# B&R Automation Studio project BatteryControl
Automation Studio 4.9.3.144 SP; technology packages: mapp 5.12.0, mappView 5.12.1

## Configuration Asfordby

CPU X20CP1381, AutomationRuntime A4.26, Build 4.1.2, Safety 0.0, Vc V4.72.2

### Hardware
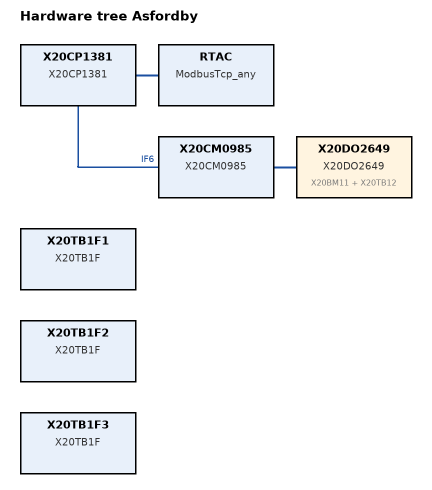
```
RTAC : ModbusTcp_any v1.0.8.0  [ETH1 -> X20CP1381.IF2 (NodeNumber=1) [Cable Type=PowerlinkCable, Length=10, Version=1.0.0.3]]
  IpAddress = 10.71.46.5
  UnitId = 1
  Cb_1
  Cb_1_FunCode = 16
  Cb_1_RefreshTime = 50
  Cb_1_SendMode = 2
  Cb_1_AddrExt = 30
  Cb_1_NumItemsExt = 2
  Cb_1_C_1
  Cb_1_C_1_Name = powerWrite
  Cb_1_C_1_Datatype = 4
  Cb_1_C_1_Dir = 1
  Cb_2
  Cb_2_FunCode = 3
  Cb_2_RefreshTime = 500
  Cb_2_Addr = 10
  Cb_2_C_1
  Cb_2_C_1_Name = operationMode
  Cb_2_C_1_Datatype = 6
  Cb_3
  Cb_3_FunCode = 6
  Cb_3_RefreshTime = 500
  Cb_3_SendMode = 2
  Cb_3_AddrExt = 28
  Cb_3_C_1
  Cb_3_C_1_Name = operationModeWrite
  Cb_3_C_1_Datatype = 6
  Cb_3_C_1_Dir = 1
  Cb_4
  Cb_4_FunCode = 3
  Cb_4_RefreshTime = 500
  Cb_4_Addr = 26
  Cb_4_C_1
  Cb_4_C_1_Name = activePower
  Cb_4_C_1_Datatype = 3
  Cb_5
  Cb_5_FunCode = 3
  Cb_5_RefreshTime = 500
  Cb_5_Addr = 20
  Cb_5_C_1
  Cb_5_C_1_Name = SOC
  Cb_5_C_1_Datatype = 6
X20BM11 : X20BM11 v1.0.0.1 (Disabled=true)  [X2X1 -> X20CM0985.X2X2]
X20CM0985 : X20CM0985 v1.0.6.1  [X2X1 -> X20CP1381.IF6]
  GenRange = 100V
  BusRange = 100V
  Sync1Range = 100V
  Sync2Range = 100V
  CurrentRange = 1A
  UnennSyn = 11000
  UnennGen = 11000
  UnennSamm = 11000
  Inenn = 1250
  Msammel = 10000
  MGen = 10000
  MSyn1 = 10000
  MSyn2 = 10000
  Mstrom = 1250
  TiefpassF = 20
  Ofrequency = 2000
  Ufrequency = 0
  Rfmin = 100
X20CP1381 : X20CP1381 v1.11.0.0  [X1 -> X1.SL; X2 -> X2.SL; X3 -> X3.SL]
  Module X1 (Type=X1, Virtual=true, Version=1.11.0.0)
    Connection (Connector=SS1, TargetModule=X20TB1F1, TargetConnector=SS)
    Connection (Connector=SL, TargetModule=X20CP1381, TargetConnector=X1)
  Module X2 (Type=X2, Virtual=true, Version=1.11.0.0)
    Connection (Connector=SS1, TargetModule=X20TB1F2, TargetConnector=SS)
    Connection (Connector=SL, TargetModule=X20CP1381, TargetConnector=X2)
  Module X3 (Type=X3, Virtual=true, Version=1.11.0.0)
    Connection (Connector=SS1, TargetModule=X20TB1F3, TargetConnector=SS)
    Connection (Connector=SL, TargetModule=X20CP1381, TargetConnector=X3)
  Connector IF2:
    ActivateDevice = 1
    Vnc1
    VncVcObjectName1 = Visu
    VncKeyMappingFile1 = VC\PS2-Keyboard.dis
    VncRefreshRate1 = 500
    VncTitle1 = Debug
    ActivateModbus = 1
    NumSlaves = -1
    NumAllBlocks = -1
    MemSizeIn = -1
    MemSizeOut = -1
  Connector IF3:
    DNAConfiguration = manual
  ConfigurationID = Static_Config1
  TimerDeviceType = SWIOTIMER
  SystemTick = 5000
  IdleTaskClass = 4
  Cyclic1Duration = 5000
  Cyclic1Tolerance = 5000
  Cyclic2Duration = 10000
  Cyclic2Tolerance = 10000
  Cyclic3Duration = 50000
  Cyclic3Tolerance = 50000
  Cyclic4Duration = 100000
  Cyclic4Tolerance = 100000
  Cyclic5Duration = 200000
  Cyclic5Tolerance = 200000
  Cyclic6Duration = 500000
  Cyclic6Tolerance = 500000
  Cyclic7Duration = 1000000
  Cyclic7Tolerance = 1000000
  Cyclic8Duration = 10000
  Cyclic8Tolerance = 30000000
  ActivateSntp = 1
  SntpcServAddr1 = 194.164.127.5
  SntpcServAddr2 = 194.164.127.4
  SntpcServAddr3 = 194.164.127.6
  SntpcServAddr4 = 81.168.77.149
  ActivateDns = 1
  DnsDefaultDomain = ukpr.local
  GetDnsFromDhcp = 2
  ActivateOpcUa = 1
  OpcUa_Security_SoftwareCertificates = 
X20DO2649 : X20DO2649 v1.1.0.0 (Disabled=true)  [SS1 -> X20TB12.SS; SL -> X20BM11.SL1]
X20TB12 : X20TB12 v1.0.0.0 (Disabled=true)
X20TB1F1 : X20TB1F v1.0.0.0
X20TB1F2 : X20TB1F v1.0.0.0
X20TB1F3 : X20TB1F v1.0.0.0
```

### IoMap.iom - X20CP1381/IoMap.iom
```iecst
VAR_CONFIG
	::operationModeWrite AT %QW."RTAC".operationModeWrite;
	::cmdOperationModeWrite AT %QX."RTAC".BlockSendOnce03;
	::OperationModeWriteACK AT %IX."RTAC".BlockSendOnceAck03;
	::RTACOperationMode AT %IW."RTAC".operationMode;
	::RTACActivePower AT %IW."RTAC".activePower;
	::RTACSoC AT %IW."RTAC".SOC;
	::DNO:DI1 AT %IX."X2a".DigitalInput01;
	::DNO:DI2 AT %IX."X2a".DigitalInput02;
	::DNO:DI3 AT %IX."X2a".DigitalInput03;
	::DNO:DO1 AT %QX."X3a".DigitalOutput01;
	::DNO:DO2 AT %QX."X3a".DigitalOutput02;
	Cyclic#2.diACSwitch AT %QX."X20DO2649".DigitalOutput01;
	aiFrequency AT %IW."X20CM0985".AnalogInput24;
	::IO:aiPF AT %IW."X20CM0985".AnalogInput23;
	::IO:aiActivePower AT %IW."X20CM0985".AnalogInput19;
	::IO:aiPhaseCurrentGenL1 AT %IW."X20CM0985".AnalogInput01;
	::IO:aiPhaseCurrentGenL2 AT %IW."X20CM0985".AnalogInput02;
	::IO:aiPhaseCurrentGenL3 AT %IW."X20CM0985".AnalogInput03;
	::IO:aiAverageCurrentGen AT %IW."X20CM0985".AnalogInput04;
	::IO:aiLineVoltageGenL1L2 AT %IW."X20CM0985".AnalogInput07;
	::IO:aiLineVoltageGenL2L3 AT %IW."X20CM0985".AnalogInput08;
	::IO:aiLineVoltageGenL3L1 AT %IW."X20CM0985".AnalogInput09;
	::IO:aiPhaseVoltageGenL1 AT %IW."X20CM0985".AnalogInput10;
	::IO:aiPhaseVoltageGenL2 AT %IW."X20CM0985".AnalogInput11;
	::IO:aiPhaseVoltageGenL3 AT %IW."X20CM0985".AnalogInput12;
	::IO:aiAverageLineVoltage AT %IW."X20CM0985".AnalogInput22;
	doACSwitch AT %QX."X20CM0985".DigitalOutput05;
	::IO:aiReactivePower AT %IW."X20CM0985".AnalogInput20;
	::IO:aiAparentPower AT %IW."X20CM0985".AnalogInput21;
	diPhase1LossGen AT %IX."X20CM0985".StatusInput12;
	::IO:aiLineVoltageBusL1L2 AT %IW."X20CM0985".AnalogInput13;
	::IO:aiLineVoltageBusL2L3 AT %IW."X20CM0985".AnalogInput14;
	::IO:aiLineVoltageBusL3L1 AT %IW."X20CM0985".AnalogInput15;
	::IO:aiPhaseVoltageL1 AT %IW."X20CM0985".AnalogInput16;
	::IO:aiPhaseVoltageL2 AT %IW."X20CM0985".AnalogInput17;
	::IO:aiPhaseVoltageL3 AT %IW."X20CM0985".AnalogInput18;
	::IO:aiLineVoltageSync1 AT %IW."X20CM0985".AnalogInput25;
	::IO:aiLineVoltageSync2 AT %IW."X20CM0985".AnalogInput26;
	::IO:aiFrequencySync1 AT %IW."X20CM0985".AnalogInput27;
	::IO:aiFrequencySync2 AT %IW."X20CM0985".AnalogInput28;
	cmdWritePowerOutput AT %QX."RTAC".BlockSendOnce01;
	WritePowerOutputACK AT %IX."RTAC".BlockSendOnceAck01;
	powerOutputDINT AT %QD."RTAC".powerWrite;
	::Modbus:RTACModuleOK AT %IX."RTAC".ModuleOk;
	::Modbus:RTACActInternalError AT %IX."RTAC".ActInternalError;
	::Modbus:RTACActContError AT %IX."RTAC".ActConfError;
	::Modbus:RTACActOverloadError AT %IX."RTAC".ActOverloadError;
	::Modbus:RTACActModusError AT %IX."RTAC".ActModbusError;
	::Modbus:RTACActSlvConError AT %IX."RTAC".ActSlvConError;
	::Modbus:RTACActRefreshError AT %IX."RTAC".ActRefreshError;
	::Modbus:RTACModSlaveState AT %IW."RTAC".ModSlaveState;
	::Modbus:RTACModbusErrorLast AT %IW."RTAC".ModbusErrorLast;
	::Modbus:RTACLastErrBlockNr AT %IW."RTAC".LastErrBlockNr;
	::Modbus:RTACModbusSlaveDiag AT %QX."RTAC".ModbusSlaveDiag;
	::Modbus:RTACModbusErrorCnt AT %IW."RTAC".ModbusErrorCnt;
	::Modbus:RTACModbusConErrorCnt AT %IW."RTAC".ModbusConErrorCnt;
	::Modbus:RTACModbusPktRefreshTimoutCnt AT %IW."RTAC".ModbusPktRefreshTimeoutCnt;
	::Modbus:RTACPktPendPerSec AT %IW."RTAC".ModbusPktPendPerSec;
	::Modbus:RTACModbusMeanResponseTime AT %IW."RTAC".ModbusMeanResponseTime;
END_VAR
```

## Configuration Percival

CPU X20CP1381, AutomationRuntime A4.26, Build 4.1.2, Vc V4.26.1, Safety 0.0

### Hardware
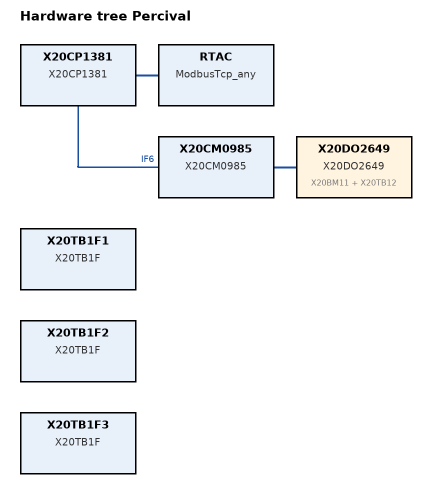
```
RTAC : ModbusTcp_any v1.0.9.0  [ETH1 -> X20CP1381.IF2 (NodeNumber=1) [Cable Type=PowerlinkCable, Length=10, Version=1.0.0.3]]
  IpAddress = 10.71.49.5
  UnitId = 1
  Cb_1
  Cb_1_FunCode = 16
  Cb_1_RefreshTime = 50
  Cb_1_SendMode = 2
  Cb_1_AddrExt = 30
  Cb_1_NumItemsExt = 2
  Cb_1_C_1
  Cb_1_C_1_Name = powerWrite
  Cb_1_C_1_Datatype = 4
  Cb_1_C_1_Dir = 1
  Cb_2
  Cb_2_FunCode = 3
  Cb_2_RefreshTime = 500
  Cb_2_Addr = 10
  Cb_2_C_1
  Cb_2_C_1_Name = operationMode
  Cb_2_C_1_Datatype = 6
  Cb_3
  Cb_3_FunCode = 6
  Cb_3_RefreshTime = 500
  Cb_3_SendMode = 2
  Cb_3_AddrExt = 28
  Cb_3_C_1
  Cb_3_C_1_Name = operationModeWrite
  Cb_3_C_1_Datatype = 6
  Cb_3_C_1_Dir = 1
  Cb_4
  Cb_4_FunCode = 3
  Cb_4_RefreshTime = 500
  Cb_4_Addr = 26
  Cb_4_C_1
  Cb_4_C_1_Name = activePower
  Cb_4_C_1_Datatype = 3
  Cb_5
  Cb_5_FunCode = 3
  Cb_5_RefreshTime = 500
  Cb_5_Addr = 20
  Cb_5_C_1
  Cb_5_C_1_Name = SOC
  Cb_5_C_1_Datatype = 6
X20BM11 : X20BM11 v1.0.0.1  [X2X1 -> X20CM0985.X2X2]
X20CM0985 : X20CM0985 v1.0.6.1  [X2X1 -> X20CP1381.IF6]
  GenRange = 100V
  BusRange = 100V
  Sync1Range = 100V
  Sync2Range = 100V
  CurrentRange = 1A
  UnennSyn = 33000
  UnennGen = 33000
  UnennSamm = 33000
  Inenn = 1250
  Msammel = 30000
  MGen = 30000
  MSyn1 = 30000
  MSyn2 = 30000
  TiefpassF = 20
  Ofrequency = 2000
  Ufrequency = 0
  Rfmin = 100
X20CP1381 : X20CP1381 v1.11.0.0  [X1 -> X1.SL; X2 -> X2.SL; X3 -> X3.SL]
  Module X1 (Type=X1, Virtual=true, Version=1.11.0.0)
    Connection (Connector=SS1, TargetModule=X20TB1F1, TargetConnector=SS)
    Connection (Connector=SL, TargetModule=X20CP1381, TargetConnector=X1)
  Module X2 (Type=X2, Virtual=true, Version=1.11.0.0)
    Connection (Connector=SS1, TargetModule=X20TB1F2, TargetConnector=SS)
    Connection (Connector=SL, TargetModule=X20CP1381, TargetConnector=X2)
  Module X3 (Type=X3, Virtual=true, Version=1.11.0.0)
    Connection (Connector=SS1, TargetModule=X20TB1F3, TargetConnector=SS)
    Connection (Connector=SL, TargetModule=X20CP1381, TargetConnector=X3)
  Connector IF2:
    ActivateDevice = 1
    Vnc1
    VncKeyMappingFile1 = VC\PS2-Keyboard.dis
    VncRefreshRate1 = 500
    VncTitle1 = Debug
    ActivateModbus = 1
    NumSlaves = -1
    NumAllBlocks = -1
    MemSizeIn = -1
    MemSizeOut = -1
  Connector IF3:
    DNAConfiguration = manual
  ConfigurationID = Static_Config1
  TimerDeviceType = SWIOTIMER
  SystemTick = 5000
  IdleTaskClass = 4
  Cyclic1Duration = 5000
  Cyclic1Tolerance = 5000
  Cyclic2Duration = 20000
  Cyclic2Tolerance = 20000
  Cyclic3Duration = 50000
  Cyclic3Tolerance = 50000
  Cyclic4Duration = 100000
  Cyclic4Tolerance = 100000
  Cyclic5Duration = 200000
  Cyclic5Tolerance = 200000
  Cyclic6Duration = 500000
  Cyclic6Tolerance = 500000
  Cyclic7Duration = 1000000
  Cyclic7Tolerance = 1000000
  Cyclic8Duration = 10000
  Cyclic8Tolerance = 30000000
  ActivateDaylightSavingTime = 1
  ActivateSntp = 1
  SntpcServAddr1 = 192.168.250.2
  ActivateDns = 1
  DnsDefaultDomain = ukpr.local
  GetDnsFromDhcp = 2
  ActivateOpcUa = 1
  OpcUa_Security_SoftwareCertificates = 
X20DO2649 : X20DO2649 v1.1.0.0  [SS1 -> X20TB12.SS; SL -> X20BM11.SL1]
X20TB12 : X20TB12 v1.0.0.0
X20TB1F1 : X20TB1F v1.0.0.0
X20TB1F2 : X20TB1F v1.0.0.0
X20TB1F3 : X20TB1F v1.0.0.0
```

### IoMap.iom - X20CP1381/IoMap.iom
```iecst
VAR_CONFIG
	::operationModeWrite AT %QW."RTAC".operationModeWrite;
	::cmdOperationModeWrite AT %QX."RTAC".BlockSendOnce03;
	::OperationModeWriteACK AT %IX."RTAC".BlockSendOnceAck03;
	::RTACOperationMode AT %IW."RTAC".operationMode;
	::RTACActivePower AT %IW."RTAC".activePower;
	::RTACSoC AT %IW."RTAC".SOC;
	::DNO:DI1 AT %IX."X2a".DigitalInput01;
	::DNO:DI2 AT %IX."X2a".DigitalInput02;
	::DNO:DI3 AT %IX."X2a".DigitalInput03;
	::DNO:DO1 AT %QX."X3a".DigitalOutput01;
	::DNO:DO2 AT %QX."X3a".DigitalOutput02;
	Cyclic#2.diACSwitch AT %QX."X20DO2649".DigitalOutput01;
	aiFrequency AT %IW."X20CM0985".AnalogInput24;
	::IO:aiPF AT %IW."X20CM0985".AnalogInput23;
	::IO:aiActivePower AT %IW."X20CM0985".AnalogInput19;
	::IO:aiPhaseCurrentGenL1 AT %IW."X20CM0985".AnalogInput01;
	::IO:aiPhaseCurrentGenL2 AT %IW."X20CM0985".AnalogInput02;
	::IO:aiPhaseCurrentGenL3 AT %IW."X20CM0985".AnalogInput03;
	::IO:aiAverageCurrentGen AT %IW."X20CM0985".AnalogInput04;
	::IO:aiLineVoltageGenL1L2 AT %IW."X20CM0985".AnalogInput07;
	::IO:aiLineVoltageGenL2L3 AT %IW."X20CM0985".AnalogInput08;
	::IO:aiLineVoltageGenL3L1 AT %IW."X20CM0985".AnalogInput09;
	::IO:aiPhaseVoltageGenL1 AT %IW."X20CM0985".AnalogInput10;
	::IO:aiPhaseVoltageGenL2 AT %IW."X20CM0985".AnalogInput11;
	::IO:aiPhaseVoltageGenL3 AT %IW."X20CM0985".AnalogInput12;
	::IO:aiAverageLineVoltage AT %IW."X20CM0985".AnalogInput22;
	doACSwitch AT %QX."X20CM0985".DigitalOutput05;
	::IO:aiReactivePower AT %IW."X20CM0985".AnalogInput20;
	::IO:aiAparentPower AT %IW."X20CM0985".AnalogInput21;
	diPhase1LossGen AT %IX."X20CM0985".StatusInput12;
	::IO:aiLineVoltageBusL1L2 AT %IW."X20CM0985".AnalogInput13;
	::IO:aiLineVoltageBusL2L3 AT %IW."X20CM0985".AnalogInput14;
	::IO:aiLineVoltageBusL3L1 AT %IW."X20CM0985".AnalogInput15;
	::IO:aiPhaseVoltageL1 AT %IW."X20CM0985".AnalogInput16;
	::IO:aiPhaseVoltageL2 AT %IW."X20CM0985".AnalogInput17;
	::IO:aiPhaseVoltageL3 AT %IW."X20CM0985".AnalogInput18;
	::IO:aiLineVoltageSync1 AT %IW."X20CM0985".AnalogInput25;
	::IO:aiLineVoltageSync2 AT %IW."X20CM0985".AnalogInput26;
	::IO:aiFrequencySync1 AT %IW."X20CM0985".AnalogInput27;
	::IO:aiFrequencySync2 AT %IW."X20CM0985".AnalogInput28;
	::powerOutputDINT AT %QD."RTAC".powerWrite;
	cmdWritePowerOutput AT %QX."RTAC".BlockSendOnce01;
	WritePowerOutputACK AT %IX."RTAC".BlockSendOnceAck01;
	::Modbus:RTACModuleOK AT %IX."RTAC".ModuleOk;
	::Modbus:RTACActInternalError AT %IX."RTAC".ActInternalError;
	::Modbus:RTACActContError AT %IX."RTAC".ActConfError;
	::Modbus:RTACActOverloadError AT %IX."RTAC".ActOverloadError;
	::Modbus:RTACActModusError AT %IX."RTAC".ActModbusError;
	::Modbus:RTACActSlvConError AT %IX."RTAC".ActSlvConError;
	::Modbus:RTACActRefreshError AT %IX."RTAC".ActRefreshError;
	::Modbus:RTACModSlaveState AT %IW."RTAC".ModSlaveState;
	::Modbus:RTACModbusErrorLast AT %IW."RTAC".ModbusErrorLast;
	::Modbus:RTACLastErrBlockNr AT %IW."RTAC".LastErrBlockNr;
	::Modbus:RTACModbusSlaveDiag AT %QX."RTAC".ModbusSlaveDiag;
	::Modbus:RTACModbusErrorCnt AT %IW."RTAC".ModbusErrorCnt;
	::Modbus:RTACModbusConErrorCnt AT %IW."RTAC".ModbusConErrorCnt;
	::Modbus:RTACModbusPktRefreshTimoutCnt AT %IW."RTAC".ModbusPktRefreshTimeoutCnt;
	::Modbus:RTACPktPendPerSec AT %IW."RTAC".ModbusPktPendPerSec;
	::Modbus:RTACModbusMeanResponseTime AT %IW."RTAC".ModbusMeanResponseTime;
END_VAR
```

## Configuration PercivalFaster

CPU X20CP1381, AutomationRuntime C4.83, Build 4.1.2, Safety 0.0, Vc V4.72.2

### Task classes (Cpu.sw)
```
Cyclic#2 (cycle 20000 us, tolerance 20000 us):
  DynamicCo1 <- DynamicContAll.prg
Cyclic#3 (cycle 50000 us, tolerance 50000 us):
  Modbus <- Modbus.prg
  RTACTest <- RTACTest.prg
  IO <- IO.prg
  StaticFFR <- StaticFFR.prg
  Manual <- Manual.prg
  DCTest <- DCTest.prg
Cyclic#4 (cycle 100000 us, tolerance 100000 us):
  Main <- Main.prg
  Settings <- Settings.prg
  VisuCtrl <- VisuCtrl.prg
Cyclic#7 (cycle 1000000 us, tolerance 1000000 us):
  Baseline <- Baseline.prg
Binaries: TCData, OpcUaMap, sysconf, Role, User, iomap, ashwd, asfw, arconfig, vcmgr, vcnet, vctcal, vcpkat, vcpdvnc, vcpfx20, Visu02, Visu03, Visu01, vccline, Visu_103, Visu_102, vccurl, vccbar, vcgclass, vcctrend, vcchtml, vccstr, vccalarm, vccovl, arial, vcpdsw, vcchspot, vccnum, vcalarm, vccdt, vccslider, vccbtn, vcfile, vccbmp, vcrt, vcshared, vcdsint, vcfntttf, vcbclass, vcdsloc, vcxml, arialbd, vcctext
Libraries: standard, MTLookUp, sys_lib, brsystem, runtime, MTFilter, MTTypes, AsBrMath, LoopCont, asieccon, astime, ashw, fileio, vcresman, dataobj
```

### Hardware
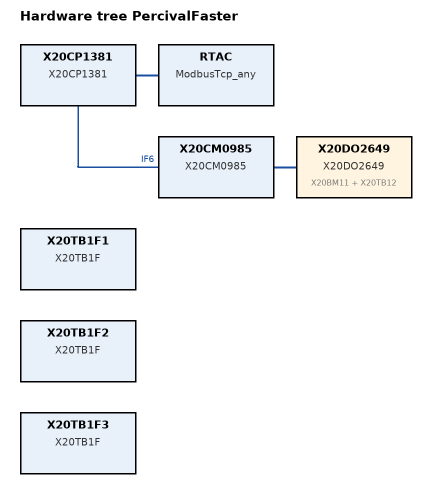
```
RTAC : ModbusTcp_any v1.0.8.0  [ETH1 -> X20CP1381.IF2 (NodeNumber=1) [Cable Type=PowerlinkCable, Length=10, Version=1.0.0.3]]
  IpAddress = 10.71.49.5
  UnitId = 1
  Cb_1
  Cb_1_FunCode = 16
  Cb_1_RefreshTime = 50
  Cb_1_SendMode = 2
  Cb_1_AddrExt = 30
  Cb_1_NumItemsExt = 2
  Cb_1_C_1
  Cb_1_C_1_Name = powerWrite
  Cb_1_C_1_Datatype = 4
  Cb_1_C_1_Dir = 1
  Cb_2
  Cb_2_FunCode = 3
  Cb_2_RefreshTime = 500
  Cb_2_Addr = 10
  Cb_2_C_1
  Cb_2_C_1_Name = operationMode
  Cb_2_C_1_Datatype = 6
  Cb_3
  Cb_3_FunCode = 6
  Cb_3_RefreshTime = 500
  Cb_3_SendMode = 2
  Cb_3_AddrExt = 28
  Cb_3_C_1
  Cb_3_C_1_Name = operationModeWrite
  Cb_3_C_1_Datatype = 6
  Cb_3_C_1_Dir = 1
  Cb_4
  Cb_4_FunCode = 3
  Cb_4_RefreshTime = 500
  Cb_4_Addr = 26
  Cb_4_C_1
  Cb_4_C_1_Name = activePower
  Cb_4_C_1_Datatype = 3
  Cb_5
  Cb_5_FunCode = 3
  Cb_5_RefreshTime = 500
  Cb_5_Addr = 20
  Cb_5_C_1
  Cb_5_C_1_Name = SOC
  Cb_5_C_1_Datatype = 6
X20BM11 : X20BM11 v1.0.0.1  [X2X1 -> X20CM0985.X2X2]
X20CM0985 : X20CM0985 v1.0.6.1  [X2X1 -> X20CP1381.IF6]
  GenRange = 100V
  BusRange = 100V
  Sync1Range = 100V
  Sync2Range = 100V
  CurrentRange = 1A
  UnennSyn = 33000
  UnennGen = 33000
  UnennSamm = 33000
  Inenn = 1250
  Msammel = 30000
  MGen = 30000
  MSyn1 = 30000
  MSyn2 = 30000
  TiefpassF = 20
  Ofrequency = 2000
  Ufrequency = 0
  Rfmin = 100
X20CP1381 : X20CP1381 v1.11.0.0  [X1 -> X1.SL; X2 -> X2.SL; X3 -> X3.SL]
  Module X1 (Type=X1, Virtual=true, Version=1.11.0.0)
    Connection (Connector=SS1, TargetModule=X20TB1F1, TargetConnector=SS)
    Connection (Connector=SL, TargetModule=X20CP1381, TargetConnector=X1)
  Module X2 (Type=X2, Virtual=true, Version=1.11.0.0)
    Connection (Connector=SS1, TargetModule=X20TB1F2, TargetConnector=SS)
    Connection (Connector=SL, TargetModule=X20CP1381, TargetConnector=X2)
  Module X3 (Type=X3, Virtual=true, Version=1.11.0.0)
    Connection (Connector=SS1, TargetModule=X20TB1F3, TargetConnector=SS)
    Connection (Connector=SL, TargetModule=X20CP1381, TargetConnector=X3)
  Connector IF2:
    ActivateDevice = 1
    Vnc1
    VncKeyMappingFile1 = VC\PS2-Keyboard.dis
    VncRefreshRate1 = 500
    VncTitle1 = Debug
    ActivateModbus = 1
    NumSlaves = -1
    NumAllBlocks = -1
    MemSizeIn = -1
    MemSizeOut = -1
  Connector IF3:
    DNAConfiguration = manual
  ConfigurationID = Static_Config1
  TimerDeviceType = SWIOTIMER
  SystemTick = 5000
  IdleTaskClass = 4
  Cyclic1Duration = 5000
  Cyclic1Tolerance = 5000
  Cyclic2Duration = 20000
  Cyclic2Tolerance = 20000
  Cyclic3Duration = 50000
  Cyclic3Tolerance = 50000
  Cyclic4Duration = 100000
  Cyclic4Tolerance = 100000
  Cyclic5Duration = 200000
  Cyclic5Tolerance = 200000
  Cyclic6Duration = 500000
  Cyclic6Tolerance = 500000
  Cyclic7Duration = 1000000
  Cyclic7Tolerance = 1000000
  Cyclic8Duration = 10000
  Cyclic8Tolerance = 30000000
  ActivateDaylightSavingTime = 1
  ActivateSntp = 1
  SntpcServAddr1 = 0.uk.pool.ntp.org
  SntpcServAddr2 = 1.uk.pool.ntp.org
  SntpcServAddr3 = 2.uk.pool.ntp.org
  SntpcServAddr4 = 3.uk.pool.ntp.org
  ActivateDns = 1
  DnsDefaultDomain = ukpr.local
  GetDnsFromDhcp = 2
  ActivateOpcUa = 1
  OpcUa_Security_SoftwareCertificates = 
X20DO2649 : X20DO2649 v1.1.0.0  [SS1 -> X20TB12.SS; SL -> X20BM11.SL1]
X20TB12 : X20TB12 v1.0.0.0
X20TB1F1 : X20TB1F v1.0.0.0
X20TB1F2 : X20TB1F v1.0.0.0
X20TB1F3 : X20TB1F v1.0.0.0
```

## Configuration SolihullTest

CPU X20CP1301, AutomationRuntime A4.26, Build 4.1.2, Vc V4.26.1, Safety 0.0

### Task classes (Cpu.sw)
```
Cyclic#2 (cycle 20000 us, tolerance 20000 us):
  IO <- IO.prg
  Modbus <- Modbus.prg
  DynamicCon <- DynamicContainment.prg
  StaticFFR <- StaticFFR.prg
  Manual <- Manual.prg
Cyclic#3 (cycle 50000 us, tolerance 50000 us):
  RTACTest <- RTACTest.prg
Cyclic#4 (cycle 100000 us, tolerance 100000 us):
  Main <- Main.prg
  Settings <- Settings.prg
  VisuCtrl <- VisuCtrl.prg
Binaries: TCData, vcctext, arialbd, vcxml, vcdsloc, vcbclass, vcfntttf, vcdsint, vcshared, vcrt, vccbmp, vcfile, vccbtn, vccslider, vccdt, vcalarm, vccnum, vcchspot, vcpdsw, arial, vccovl, vccalarm, vccstr, vcchtml, vcctrend, vcgclass, vccbar, vccurl, Visu_102, Visu_103, OpcUaMap, sysconf, Role, User, iomap, ashwd, asfw, arconfig, vccline, Visu01, Visu03, Visu02, vcpfx20, vcpdvnc, vcpkat, vctcal, vcnet, vcmgr
Libraries: standard, astime, asieccon, MTLookUp, sys_lib, brsystem, runtime, dataobj, vcresman, fileio, MTFilter, MTTypes, AsBrMath, ashw
```

### Hardware
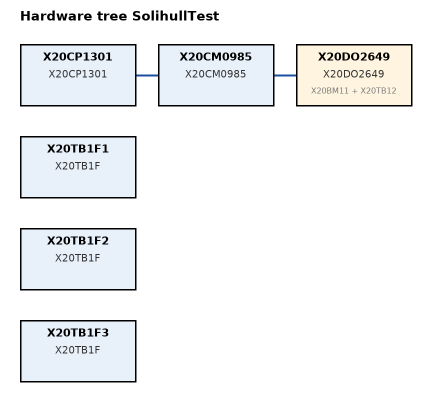
```
X20BM11 : X20BM11 v1.0.0.1  [X2X1 -> X20CM0985.X2X2]
X20CM0985 : X20CM0985 v1.0.6.1  [X2X1 -> X20CP1301.IF6]
  Supervision = off
  GenRange = 100V
  BusRange = 100V
  Sync1Range = 100V
  Sync2Range = 100V
  CurrentRange = 1A
  UnennSyn = 33000
  UnennGen = 33000
  UnennSamm = 33000
  Inenn = 1250
  Msammel = 30000
  MGen = 30000
  MSyn1 = 30000
  MSyn2 = 30000
  Ofrequency = 2000
  Ufrequency = 0
  Rfmin = 100
X20CP1301 : X20CP1301 v1.3.0.0  [X1 -> X1.SL; X2 -> X2.SL; X3 -> X3.SL]
  Module X1 (Type=X1, Virtual=true, Version=1.0.0.0)
    Connection (Connector=SS1, TargetModule=X20TB1F1, TargetConnector=SS)
    Connection (Connector=SL, TargetModule=X20CP1301, TargetConnector=X1)
  Module X2 (Type=X2, Virtual=true, Version=1.0.0.0)
    Connection (Connector=SS1, TargetModule=X20TB1F2, TargetConnector=SS)
    Connection (Connector=SL, TargetModule=X20CP1301, TargetConnector=X2)
  Module X3 (Type=X3, Virtual=true, Version=1.0.0.0)
    Connection (Connector=SS1, TargetModule=X20TB1F3, TargetConnector=SS)
    Connection (Connector=SL, TargetModule=X20CP1301, TargetConnector=X3)
  Connector IF2:
    ActivateDevice = 1
    Vnc1
    VncKeyMappingFile1 = VC\PS2-Keyboard.dis
    VncRefreshRate1 = 500
    VncTitle1 = Debug
    ActivateModbus = 1
    NumSlaves = -1
    NumAllBlocks = -1
    MemSizeIn = -1
    MemSizeOut = -1
  ConfigurationID = Static_Config1
  TimerDeviceType = SWIOTIMER
  SystemTick = 5000
  IdleTaskClass = 4
  Cyclic1Duration = 5000
  Cyclic1Tolerance = 5000
  Cyclic2Duration = 20000
  Cyclic2Tolerance = 20000
  Cyclic3Duration = 50000
  Cyclic3Tolerance = 50000
  Cyclic4Duration = 100000
  Cyclic4Tolerance = 100000
  Cyclic5Duration = 200000
  Cyclic5Tolerance = 200000
  Cyclic6Duration = 500000
  Cyclic6Tolerance = 500000
  Cyclic7Duration = 1000000
  Cyclic7Tolerance = 1000000
  Cyclic8Duration = 10000
  Cyclic8Tolerance = 30000000
  ActivateDaylightSavingTime = 1
  ActivateSntp = 1
  SntpcServAddr1 = 194.164.127.5
  SntpcServAddr2 = 194.164.127.4
  SntpcServAddr3 = 194.164.127.6
  SntpcServAddr4 = 81.168.77.149
  ActivateDns = 1
  DnsDefaultDomain = ukpr.local
  GetDnsFromDhcp = 2
  DCOMInterface = IF2
  ActivateOpcUa = 1
  OpcUa_Security_SoftwareCertificates = 
X20DO2649 : X20DO2649 v1.0.2.0  [SS1 -> X20TB12.SS; SL -> X20BM11.SL1]
  Supervision = off
X20TB12 : X20TB12 v1.0.0.0
X20TB1F1 : X20TB1F v1.0.0.0
X20TB1F2 : X20TB1F v1.0.0.0
X20TB1F3 : X20TB1F v1.0.0.0
```

### IoMap.iom - X20CP1301/IoMap.iom
```iecst
VAR_CONFIG
	::DNO:DI1 AT %IX."X2a".DigitalInput01;
	::DNO:DI2 AT %IX."X2a".DigitalInput02;
	::DNO:DI3 AT %IX."X2a".DigitalInput03;
	::DNO:DO1 AT %QX."X3a".DigitalOutput01;
	::DNO:DO2 AT %QX."X3a".DigitalOutput02;
	Cyclic#2.diACSwitch AT %QX."X20DO2649".DigitalOutput01;
	aiFrequency AT %IW."X20CM0985".AnalogInput24;
	::IO:aiPF AT %IW."X20CM0985".AnalogInput23;
	::IO:aiActivePower AT %IW."X20CM0985".AnalogInput19;
	::IO:aiPhaseCurrentGenL1 AT %IW."X20CM0985".AnalogInput01;
	::IO:aiPhaseCurrentGenL2 AT %IW."X20CM0985".AnalogInput02;
	::IO:aiPhaseCurrentGenL3 AT %IW."X20CM0985".AnalogInput03;
	::IO:aiAverageCurrentGen AT %IW."X20CM0985".AnalogInput04;
	::IO:aiLineVoltageGenL1L2 AT %IW."X20CM0985".AnalogInput07;
	::IO:aiLineVoltageGenL2L3 AT %IW."X20CM0985".AnalogInput08;
	::IO:aiLineVoltageGenL3L1 AT %IW."X20CM0985".AnalogInput09;
	::IO:aiPhaseVoltageGenL1 AT %IW."X20CM0985".AnalogInput10;
	::IO:aiPhaseVoltageGenL2 AT %IW."X20CM0985".AnalogInput11;
	::IO:aiPhaseVoltageGenL3 AT %IW."X20CM0985".AnalogInput12;
	::IO:aiAverageLineVoltage AT %IW."X20CM0985".AnalogInput22;
	doACSwitch AT %QX."X20CM0985".DigitalOutput05;
	::IO:aiReactivePower AT %IW."X20CM0985".AnalogInput20;
	::IO:aiAparentPower AT %IW."X20CM0985".AnalogInput21;
	diPhase1LossGen AT %IX."X20CM0985".StatusInput12;
	::IO:aiLineVoltageBusL1L2 AT %IW."X20CM0985".AnalogInput13;
	::IO:aiLineVoltageBusL2L3 AT %IW."X20CM0985".AnalogInput14;
	::IO:aiLineVoltageBusL3L1 AT %IW."X20CM0985".AnalogInput15;
	::IO:aiPhaseVoltageL1 AT %IW."X20CM0985".AnalogInput16;
	::IO:aiPhaseVoltageL2 AT %IW."X20CM0985".AnalogInput17;
	::IO:aiPhaseVoltageL3 AT %IW."X20CM0985".AnalogInput18;
	::IO:aiLineVoltageSync1 AT %IW."X20CM0985".AnalogInput25;
	::IO:aiLineVoltageSync2 AT %IW."X20CM0985".AnalogInput26;
	::IO:aiFrequencySync1 AT %IW."X20CM0985".AnalogInput27;
	::IO:aiFrequencySync2 AT %IW."X20CM0985".AnalogInput28;
END_VAR
```

## Configuration SolihullTest2

CPU X20CP1382, AutomationRuntime A4.26, Build 4.1.2, Vc V4.26.1, Safety 0.0

### Task classes (Cpu.sw)
```
Cyclic#3 (cycle 50000 us, tolerance 50000 us):
  RTACTest <- RTACTest.prg
  IO <- IO.prg
  Modbus <- Modbus.prg
  DynamicCon <- DynamicContainment.prg
  StaticFFR <- StaticFFR.prg
  Manual <- Manual.prg
Cyclic#4 (cycle 100000 us, tolerance 100000 us):
  Main <- Main.prg
  Settings <- Settings.prg
  VisuCtrl <- VisuCtrl.prg
VcDataObjects: Visu <- Visu.dob
Binaries: TCData, vcctext, arialbd, vcmgr, vcxml, vcnet, Visu02, vcdsloc, vcbclass, vcfntttf, vcdsint, vctcal, Visu03, vcshared, vcrt, vcpkat, Visu01, vccbmp, vcfile, vccbtn, vccslider, vccdt, vcalarm, vccnum, vcchspot, vcpdsw, arial, vccovl, vccalarm, vcpdvnc, vccstr, vcchtml, vcctrend, vcgclass, vccbar, vccurl, vcpfx20, arconfig, asfw, ashwd, iomap, User, Role, sysconf, OpcUaMap, vccline
Libraries: standard, astime, asieccon, MTLookUp, sys_lib, brsystem, runtime, ashw, dataobj, vcresman, fileio, MTFilter, MTTypes, AsBrMath
```

### Hardware
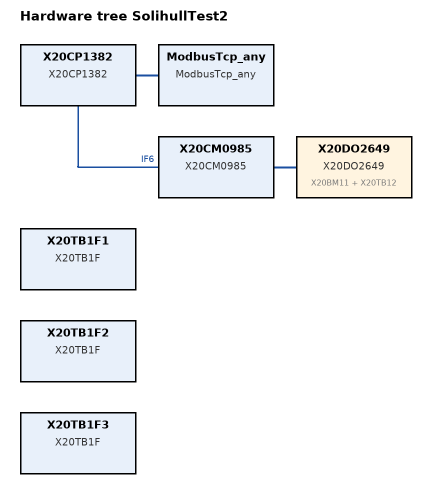
```
ModbusTcp_any : ModbusTcp_any v1.0.9.0  [ETH1 -> X20CP1382.IF2 (NodeNumber=1) [Cable Type=PowerlinkCable, Length=10, Version=1.0.0.3]]
  IpAddress = 10.71.46.5
  UnitId = 1
  Cb_1
  Cb_1_FunCode = 6
  Cb_1_RefreshTime = 20
  Cb_1_SendMode = 2
  Cb_1_AddrExt = 30
  Cb_1_C_1
  Cb_1_C_1_Name = powerWrite
  Cb_1_C_1_Datatype = 3
  Cb_1_C_1_Dir = 1
  Cb_2
  Cb_2_FunCode = 3
  Cb_2_RefreshTime = 20
  Cb_2_Addr = 10
  Cb_2_C_1
  Cb_2_C_1_Name = operationMode
  Cb_2_C_1_Datatype = 6
  Cb_3
  Cb_3_FunCode = 6
  Cb_3_RefreshTime = 20
  Cb_3_SendMode = 2
  Cb_3_AddrExt = 28
  Cb_3_C_1
  Cb_3_C_1_Name = operationModeWrite
  Cb_3_C_1_Datatype = 6
  Cb_3_C_1_Dir = 1
  Cb_4
  Cb_4_FunCode = 3
  Cb_4_RefreshTime = 20
  Cb_4_Addr = 26
  Cb_4_C_1
  Cb_4_C_1_Name = activePower
  Cb_4_C_1_Datatype = 3
  Cb_5
  Cb_5_FunCode = 3
  Cb_5_RefreshTime = 20
  Cb_5_Addr = 20
  Cb_5_C_1
  Cb_5_C_1_Name = SOC
  Cb_5_C_1_Datatype = 6
X20BM11 : X20BM11 v1.0.0.1 (Disabled=true)  [X2X1 -> X20CM0985.X2X2]
X20CM0985 : X20CM0985 v1.0.6.1  [X2X1 -> X20CP1382.IF6]
  GenRange = 100V
  BusRange = 100V
  Sync1Range = 100V
  Sync2Range = 100V
  CurrentRange = 1A
  UnennSyn = 11000
  UnennGen = 11000
  UnennSamm = 11000
  Inenn = 1250
  Msammel = 10000
  MGen = 10000
  MSyn1 = 10000
  MSyn2 = 10000
  Mstrom = 1250
  Ofrequency = 2000
  Ufrequency = 0
  Rfmin = 100
X20CP1382 : X20CP1382 v1.11.0.0  [X1 -> X1a.SL; X2 -> X2a.SL; X3 -> X3a.SL]
  Module X1a (Type=X1, Virtual=true, Version=1.11.0.0)
    Connection (Connector=SS1, TargetModule=X20TB1F1, TargetConnector=SS)
    Connection (Connector=SL, TargetModule=X20CP1382, TargetConnector=X1)
  Module X2a (Type=X2, Virtual=true, Version=1.11.0.0)
    Connection (Connector=SS1, TargetModule=X20TB1F2, TargetConnector=SS)
    Connection (Connector=SL, TargetModule=X20CP1382, TargetConnector=X2)
  Module X3a (Type=X3, Virtual=true, Version=1.11.0.0)
    Connection (Connector=SS1, TargetModule=X20TB1F3, TargetConnector=SS)
    Connection (Connector=SL, TargetModule=X20CP1382, TargetConnector=X3)
  Connector IF2:
    ActivateDevice = 1
    Vnc1
    VncVcObjectName1 = Visu
    VncKeyMappingFile1 = VC\PS2-Keyboard.dis
    VncRefreshRate1 = 500
    VncTitle1 = Debug
    ActivateModbus = 1
    NumSlaves = -1
    NumAllBlocks = -1
    MemSizeIn = -1
    MemSizeOut = -1
  Connector IF3:
    DNAConfiguration = manual
  ConfigurationID = Static_Config1
  TimerDeviceType = SWIOTIMER
  SystemTick = 5000
  IdleTaskClass = 4
  Cyclic1Duration = 5000
  Cyclic1Tolerance = 5000
  Cyclic2Duration = 20000
  Cyclic2Tolerance = 20000
  Cyclic3Duration = 50000
  Cyclic3Tolerance = 50000
  Cyclic4Duration = 100000
  Cyclic4Tolerance = 100000
  Cyclic5Duration = 200000
  Cyclic5Tolerance = 200000
  Cyclic6Duration = 500000
  Cyclic6Tolerance = 500000
  Cyclic7Duration = 1000000
  Cyclic7Tolerance = 1000000
  Cyclic8Duration = 10000
  Cyclic8Tolerance = 30000000
  ActivateSntp = 1
  SntpcServAddr1 = 194.164.127.5
  SntpcServAddr2 = 194.164.127.4
  SntpcServAddr3 = 194.164.127.6
  SntpcServAddr4 = 81.168.77.149
  ActivateDns = 1
  DnsDefaultDomain = ukpr.local
  GetDnsFromDhcp = 2
  ActivateOpcUa = 1
  OpcUa_Security_SoftwareCertificates = 
X20DO2649 : X20DO2649 v1.1.0.0 (Disabled=true)  [SS1 -> X20TB12.SS; SL -> X20BM11.SL1]
X20TB12 : X20TB12 v1.0.0.0 (Disabled=true)
X20TB1F1 : X20TB1F v1.0.0.0
X20TB1F2 : X20TB1F v1.0.0.0
X20TB1F3 : X20TB1F v1.0.0.0
```

### IoMap.iom - X20CP1382/IoMap.iom
```iecst
VAR_CONFIG
	Cyclic#2.::powerOutput AT %QW."ModbusTcp_any".powerWrite;
	::operationModeWrite AT %QW."ModbusTcp_any".operationModeWrite;
	::cmdOperationModeWrite AT %QX."ModbusTcp_any".BlockSendOnce03;
	::OperationModeWriteACK AT %IX."ModbusTcp_any".BlockSendOnceAck03;
	::RTACOperationMode AT %IW."ModbusTcp_any".operationMode;
	::RTACActivePower AT %IW."ModbusTcp_any".activePower;
	::RTACSoC AT %IW."ModbusTcp_any".SOC;
	::DNO:DI1 AT %IX."X2a".DigitalInput01;
	::DNO:DI2 AT %IX."X2a".DigitalInput02;
	::DNO:DI3 AT %IX."X2a".DigitalInput03;
	::DNO:DO1 AT %QX."X3a".DigitalOutput01;
	::DNO:DO2 AT %QX."X3a".DigitalOutput02;
	Cyclic#2.diACSwitch AT %QX."X20DO2649".DigitalOutput01;
	cmdWritePowerOutput AT %QX."ModbusTcp_any".BlockSendOnce01;
	WritePowerOutputACK AT %IX."ModbusTcp_any".BlockSendOnceAck01;
	aiFrequency AT %IW."X20CM0985".AnalogInput24;
	::IO:aiPF AT %IW."X20CM0985".AnalogInput23;
	::IO:aiActivePower AT %IW."X20CM0985".AnalogInput19;
	::IO:aiPhaseCurrentGenL1 AT %IW."X20CM0985".AnalogInput01;
	::IO:aiPhaseCurrentGenL2 AT %IW."X20CM0985".AnalogInput02;
	::IO:aiPhaseCurrentGenL3 AT %IW."X20CM0985".AnalogInput03;
	::IO:aiAverageCurrentGen AT %IW."X20CM0985".AnalogInput04;
	::IO:aiLineVoltageGenL1L2 AT %IW."X20CM0985".AnalogInput07;
	::IO:aiLineVoltageGenL2L3 AT %IW."X20CM0985".AnalogInput08;
	::IO:aiLineVoltageGenL3L1 AT %IW."X20CM0985".AnalogInput09;
	::IO:aiPhaseVoltageGenL1 AT %IW."X20CM0985".AnalogInput10;
	::IO:aiPhaseVoltageGenL2 AT %IW."X20CM0985".AnalogInput11;
	::IO:aiPhaseVoltageGenL3 AT %IW."X20CM0985".AnalogInput12;
	::IO:aiAverageLineVoltage AT %IW."X20CM0985".AnalogInput22;
	doACSwitch AT %QX."X20CM0985".DigitalOutput05;
	::IO:aiReactivePower AT %IW."X20CM0985".AnalogInput20;
	::IO:aiAparentPower AT %IW."X20CM0985".AnalogInput21;
	diPhase1LossGen AT %IX."X20CM0985".StatusInput12;
	::IO:aiLineVoltageBusL1L2 AT %IW."X20CM0985".AnalogInput13;
	::IO:aiLineVoltageBusL2L3 AT %IW."X20CM0985".AnalogInput14;
	::IO:aiLineVoltageBusL3L1 AT %IW."X20CM0985".AnalogInput15;
	::IO:aiPhaseVoltageL1 AT %IW."X20CM0985".AnalogInput16;
	::IO:aiPhaseVoltageL2 AT %IW."X20CM0985".AnalogInput17;
	::IO:aiPhaseVoltageL3 AT %IW."X20CM0985".AnalogInput18;
	::IO:aiLineVoltageSync1 AT %IW."X20CM0985".AnalogInput25;
	::IO:aiLineVoltageSync2 AT %IW."X20CM0985".AnalogInput26;
	::IO:aiFrequencySync1 AT %IW."X20CM0985".AnalogInput27;
	::IO:aiFrequencySync2 AT %IW."X20CM0985".AnalogInput28;
END_VAR
```

## Configuration Vauxhall

CPU X20CP1382, AutomationRuntime C4.83, Build 4.1.2, Safety 0.0, Vc V4.72.2

### Task classes (Cpu.sw)
```
Cyclic#3 (cycle 50000 us, tolerance 50000 us):
  Modbus <- Modbus.prg
  RTACTest <- RTACTest.prg
  IO <- IO.prg
  DynamicCon <- DynamicContainment.prg
  StaticFFR <- StaticFFR.prg
  Manual <- Manual.prg
  DCTest <- DCTest.prg
Cyclic#4 (cycle 100000 us, tolerance 100000 us):
  Main <- Main.prg
  Settings <- Settings.prg
  VisuCtrl <- VisuCtrl.prg
Cyclic#7 (cycle 1000000 us, tolerance 1000000 us):
  Baseline <- Baseline.prg
Binaries: TCData, OpcUaMap, sysconf, Role, User, iomap, ashwd, asfw, arconfig, vcctext, arialbd, vcxml, vcdsloc, vcbclass, vcfntttf, vcdsint, vcshared, vcrt, vccbmp, vcfile, vccbtn, vccslider, vccdt, vcalarm, vccnum, vcchspot, vcpdsw, arial, vccovl, vccalarm, vccstr, vcchtml, vcctrend, vcgclass, vccbar, vccurl, Visu_102, Visu_103, vccline, Visu01, Visu03, Visu02, vcpfx20, vcpdvnc, vcpkat, vctcal, vcnet, vcmgr
Libraries: standard, astime, asieccon, MTLookUp, sys_lib, brsystem, runtime, MTFilter, MTTypes, AsBrMath, LoopCont, dataobj, vcresman, fileio, ashw
```

### Hardware
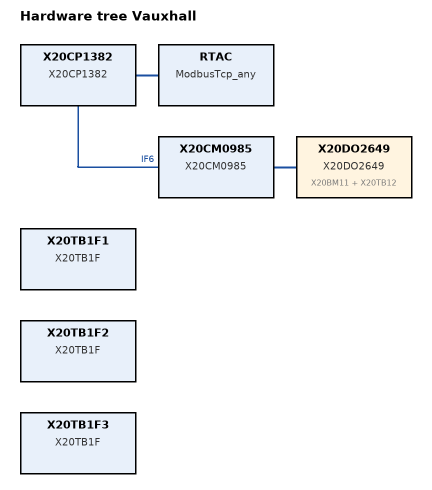
```
RTAC : ModbusTcp_any v1.0.8.0  [ETH1 -> X20CP1382.IF2 (NodeNumber=1) [Cable Type=PowerlinkCable, Length=10, Version=1.0.0.3]]
  IpAddress = 10.71.50.5
  UnitId = 1
  Cb_1
  Cb_1_FunCode = 16
  Cb_1_RefreshTime = 50
  Cb_1_SendMode = 2
  Cb_1_AddrExt = 30
  Cb_1_NumItemsExt = 2
  Cb_1_C_1
  Cb_1_C_1_Name = powerWrite
  Cb_1_C_1_Datatype = 4
  Cb_1_C_1_Dir = 1
  Cb_2
  Cb_2_FunCode = 3
  Cb_2_RefreshTime = 500
  Cb_2_Addr = 10
  Cb_2_C_1
  Cb_2_C_1_Name = operationMode
  Cb_2_C_1_Datatype = 6
  Cb_3
  Cb_3_FunCode = 6
  Cb_3_RefreshTime = 500
  Cb_3_SendMode = 2
  Cb_3_AddrExt = 28
  Cb_3_C_1
  Cb_3_C_1_Name = operationModeWrite
  Cb_3_C_1_Datatype = 6
  Cb_3_C_1_Dir = 1
  Cb_4
  Cb_4_FunCode = 3
  Cb_4_RefreshTime = 500
  Cb_4_Addr = 26
  Cb_4_C_1
  Cb_4_C_1_Name = activePower
  Cb_4_C_1_Datatype = 3
  Cb_5
  Cb_5_FunCode = 3
  Cb_5_RefreshTime = 500
  Cb_5_Addr = 20
  Cb_5_C_1
  Cb_5_C_1_Name = SOC
  Cb_5_C_1_Datatype = 6
X20BM11 : X20BM11 v1.0.0.1 (Disabled=true)  [X2X1 -> X20CM0985.X2X2]
X20CM0985 : X20CM0985 v1.0.6.1  [X2X1 -> X20CP1382.IF6]
  GenRange = 100V
  BusRange = 100V
  Sync1Range = 100V
  Sync2Range = 100V
  CurrentRange = 1A
  UnennSyn = 33000
  UnennGen = 33000
  UnennSamm = 33000
  Inenn = 1250
  Msammel = 30000
  MGen = 30000
  MSyn1 = 30000
  MSyn2 = 30000
  TiefpassF = 20
  Ofrequency = 2000
  Ufrequency = 0
  Rfmin = 100
X20CP1382 : X20CP1382 v1.11.0.0  [X1 -> X1.SL; X2 -> X2.SL; X3 -> X3.SL]
  Module X1 (Type=X1, Virtual=true, Version=1.11.0.0)
    Connection (Connector=SS1, TargetModule=X20TB1F1, TargetConnector=SS)
    Connection (Connector=SL, TargetModule=X20CP1382, TargetConnector=X1)
  Module X2 (Type=X2, Virtual=true, Version=1.11.0.0)
    Connection (Connector=SS1, TargetModule=X20TB1F2, TargetConnector=SS)
    Connection (Connector=SL, TargetModule=X20CP1382, TargetConnector=X2)
  Module X3 (Type=X3, Virtual=true, Version=1.11.0.0)
    Connection (Connector=SS1, TargetModule=X20TB1F3, TargetConnector=SS)
    Connection (Connector=SL, TargetModule=X20CP1382, TargetConnector=X3)
  Connector IF2:
    ActivateDevice = 1
    Vnc1
    VncKeyMappingFile1 = VC\PS2-Keyboard.dis
    VncRefreshRate1 = 500
    VncTitle1 = Debug
    ActivateModbus = 1
    NumSlaves = -1
    NumAllBlocks = -1
    MemSizeIn = -1
    MemSizeOut = -1
  Connector IF3:
    DNAConfiguration = manual
  ConfigurationID = Static_Config1
  PermanentPvSize = 4096
  TimerDeviceType = SWIOTIMER
  SystemTick = 5000
  IdleTaskClass = 4
  Cyclic1Duration = 5000
  Cyclic1Tolerance = 5000
  Cyclic2Duration = 20000
  Cyclic2Tolerance = 20000
  Cyclic3Duration = 50000
  Cyclic3Tolerance = 50000
  Cyclic4Duration = 100000
  Cyclic4Tolerance = 100000
  Cyclic5Duration = 200000
  Cyclic5Tolerance = 200000
  Cyclic6Duration = 500000
  Cyclic6Tolerance = 500000
  Cyclic7Duration = 1000000
  Cyclic7Tolerance = 1000000
  Cyclic8Duration = 10000
  Cyclic8Tolerance = 30000000
  ActivateDaylightSavingTime = 1
  ActivateSntp = 1
  SntpcServAddr1 = 0.uk.pool.ntp.org
  SntpcServAddr2 = 1.uk.pool.ntp.org
  SntpcServAddr3 = 2.uk.pool.ntp.org
  SntpcServAddr4 = 3.uk.pool.ntp.org
  ActivateDns = 1
  DnsDefaultDomain = ukpr.local
  GetDnsFromDhcp = 2
  ActivateOpcUa = 1
  OpcUa_Security_SoftwareCertificates = 
X20DO2649 : X20DO2649 v1.1.0.0 (Disabled=true)  [SS1 -> X20TB12.SS; SL -> X20BM11.SL1]
X20TB12 : X20TB12 v1.0.0.0 (Disabled=true)
X20TB1F1 : X20TB1F v1.0.0.0
X20TB1F2 : X20TB1F v1.0.0.0
X20TB1F3 : X20TB1F v1.0.0.0
```

### IoMap.iom - X20CP1382/IoMap.iom
```iecst
VAR_CONFIG
	::operationModeWrite AT %QW."RTAC".operationModeWrite;
	::cmdOperationModeWrite AT %QX."RTAC".BlockSendOnce03;
	::OperationModeWriteACK AT %IX."RTAC".BlockSendOnceAck03;
	::RTACOperationMode AT %IW."RTAC".operationMode;
	::RTACActivePower AT %IW."RTAC".activePower;
	::RTACSoC AT %IW."RTAC".SOC;
	::DNO:DI1 AT %IX."X2a".DigitalInput01;
	::DNO:DI2 AT %IX."X2a".DigitalInput02;
	::DNO:DI3 AT %IX."X2a".DigitalInput03;
	::DNO:DO1 AT %QX."X3a".DigitalOutput01;
	::DNO:DO2 AT %QX."X3a".DigitalOutput02;
	Cyclic#2.diACSwitch AT %QX."X20DO2649".DigitalOutput01;
	aiFrequency AT %IW."X20CM0985".AnalogInput24;
	::IO:aiPF AT %IW."X20CM0985".AnalogInput23;
	::IO:aiActivePower AT %IW."X20CM0985".AnalogInput19;
	::IO:aiPhaseCurrentGenL1 AT %IW."X20CM0985".AnalogInput01;
	::IO:aiPhaseCurrentGenL2 AT %IW."X20CM0985".AnalogInput02;
	::IO:aiPhaseCurrentGenL3 AT %IW."X20CM0985".AnalogInput03;
	::IO:aiAverageCurrentGen AT %IW."X20CM0985".AnalogInput04;
	::IO:aiLineVoltageGenL1L2 AT %IW."X20CM0985".AnalogInput07;
	::IO:aiLineVoltageGenL2L3 AT %IW."X20CM0985".AnalogInput08;
	::IO:aiLineVoltageGenL3L1 AT %IW."X20CM0985".AnalogInput09;
	::IO:aiPhaseVoltageGenL1 AT %IW."X20CM0985".AnalogInput10;
	::IO:aiPhaseVoltageGenL2 AT %IW."X20CM0985".AnalogInput11;
	::IO:aiPhaseVoltageGenL3 AT %IW."X20CM0985".AnalogInput12;
	::IO:aiAverageLineVoltage AT %IW."X20CM0985".AnalogInput22;
	doACSwitch AT %QX."X20CM0985".DigitalOutput05;
	::IO:aiReactivePower AT %IW."X20CM0985".AnalogInput20;
	::IO:aiAparentPower AT %IW."X20CM0985".AnalogInput21;
	diPhase1LossGen AT %IX."X20CM0985".StatusInput12;
	::IO:aiLineVoltageBusL1L2 AT %IW."X20CM0985".AnalogInput13;
	::IO:aiLineVoltageBusL2L3 AT %IW."X20CM0985".AnalogInput14;
	::IO:aiLineVoltageBusL3L1 AT %IW."X20CM0985".AnalogInput15;
	::IO:aiPhaseVoltageL1 AT %IW."X20CM0985".AnalogInput16;
	::IO:aiPhaseVoltageL2 AT %IW."X20CM0985".AnalogInput17;
	::IO:aiPhaseVoltageL3 AT %IW."X20CM0985".AnalogInput18;
	::IO:aiLineVoltageSync1 AT %IW."X20CM0985".AnalogInput25;
	::IO:aiLineVoltageSync2 AT %IW."X20CM0985".AnalogInput26;
	::IO:aiFrequencySync1 AT %IW."X20CM0985".AnalogInput27;
	::IO:aiFrequencySync2 AT %IW."X20CM0985".AnalogInput28;
	::powerOutputDINT AT %QD."RTAC".powerWrite;
	cmdWritePowerOutput AT %QX."RTAC".BlockSendOnce01;
	WritePowerOutputACK AT %IX."RTAC".BlockSendOnceAck01;
	::Modbus:RTACModuleOK AT %IX."RTAC".ModuleOk;
	::Modbus:RTACActInternalError AT %IX."RTAC".ActInternalError;
	::Modbus:RTACActContError AT %IX."RTAC".ActConfError;
	::Modbus:RTACActOverloadError AT %IX."RTAC".ActOverloadError;
	::Modbus:RTACActModusError AT %IX."RTAC".ActModbusError;
	::Modbus:RTACActSlvConError AT %IX."RTAC".ActSlvConError;
	::Modbus:RTACActRefreshError AT %IX."RTAC".ActRefreshError;
	::Modbus:RTACModSlaveState AT %IW."RTAC".ModSlaveState;
	::Modbus:RTACModbusErrorLast AT %IW."RTAC".ModbusErrorLast;
	::Modbus:RTACLastErrBlockNr AT %IW."RTAC".LastErrBlockNr;
	::Modbus:RTACModbusErrorCnt AT %IW."RTAC".ModbusErrorCnt;
	::Modbus:RTACModbusConErrorCnt AT %IW."RTAC".ModbusConErrorCnt;
	::Modbus:RTACModbusPktRefreshTimoutCnt AT %IW."RTAC".ModbusPktRefreshTimeoutCnt;
	::Modbus:RTACPktPendPerSec AT %IW."RTAC".ModbusPktPendPerSec;
	::Modbus:RTACModbusMeanResponseTime AT %IW."RTAC".ModbusMeanResponseTime;
	::Modbus:RTACModbusSlaveDiag AT %QX."RTAC".ModbusSlaveDiag;
END_VAR
```

## Configuration batlane

CPU X20CP1382, AutomationRuntime C4.83, Build 4.1.2, Safety 0.0, Vc V4.72.2

### Hardware
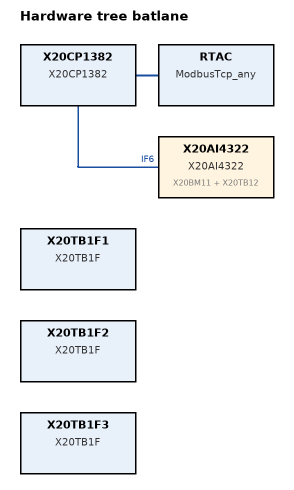
```
RTAC : ModbusTcp_any v1.0.8.0  [ETH1 -> X20CP1382.IF2 (NodeNumber=1) [Cable Type=PowerlinkCable, Length=10, Version=1.0.0.3]]
  IpAddress = 172.18.219.99
  UnitId = 1
  Cb_1
  Cb_1_FunCode = 16
  Cb_1_RefreshTime = 50
  Cb_1_SendMode = 2
  Cb_1_AddrExt = 30
  Cb_1_NumItemsExt = 2
  Cb_1_C_1
  Cb_1_C_1_Name = powerWrite
  Cb_1_C_1_Datatype = 4
  Cb_1_C_1_Dir = 1
  Cb_2
  Cb_2_FunCode = 3
  Cb_2_RefreshTime = 500
  Cb_2_Addr = 10
  Cb_2_C_1
  Cb_2_C_1_Name = operationMode
  Cb_2_C_1_Datatype = 6
  Cb_3
  Cb_3_FunCode = 6
  Cb_3_RefreshTime = 500
  Cb_3_SendMode = 2
  Cb_3_AddrExt = 28
  Cb_3_C_1
  Cb_3_C_1_Name = operationModeWrite
  Cb_3_C_1_Datatype = 6
  Cb_3_C_1_Dir = 1
  Cb_4
  Cb_4_FunCode = 3
  Cb_4_RefreshTime = 500
  Cb_4_Addr = 26
  Cb_4_C_1
  Cb_4_C_1_Name = activePower
  Cb_4_C_1_Datatype = 3
  Cb_5
  Cb_5_FunCode = 3
  Cb_5_RefreshTime = 500
  Cb_5_Addr = 20
  Cb_5_C_1
  Cb_5_C_1_Name = SOC
  Cb_5_C_1_Datatype = 6
  Cb_6
  Cb_6_FunCode = 16
  Cb_6_RefreshTime = 500
  Cb_6_AddrExt = 7580
  Cb_6_NumItemsExt = 2
  Cb_6_C_1
  Cb_6_C_1_Name = MDU_Lofreq_Full_delivery_bp
  Cb_6_C_1_Datatype = 4
  Cb_6_C_1_Dir = 1
X20AI4322 : X20AI4322 v1.1.0.0  [SS1 -> X20TB12a.SS; SL -> X20BM11a.SL1]
X20BM11a : X20BM11 v1.0.0.1  [X2X1 -> X20CP1382.IF6]
X20CP1382 : X20CP1382 v1.11.0.0  [X1 -> X1.SL; X2 -> X2.SL; X3 -> X3.SL]  //  jyh
  Module X1 (Type=X1, Virtual=true, Version=1.11.0.0)
    Connection (Connector=SS1, TargetModule=X20TB1F1, TargetConnector=SS)
    Connection (Connector=SL, TargetModule=X20CP1382, TargetConnector=X1)
  Module X2 (Type=X2, Virtual=true, Version=1.11.0.0)
    Connection (Connector=SS1, TargetModule=X20TB1F2, TargetConnector=SS)
    Connection (Connector=SL, TargetModule=X20CP1382, TargetConnector=X2)
  Module X3 (Type=X3, Virtual=true, Version=1.11.0.0)
    Connection (Connector=SS1, TargetModule=X20TB1F3, TargetConnector=SS)
    Connection (Connector=SL, TargetModule=X20CP1382, TargetConnector=X3)
  Connector IF2:
    ActivateDevice = 1
    Mode = Manual
    InternetAddress = 172.18.219.52
    SubnetMask = 255.255.255.240
    InaNodeNumber = 0
    Vnc1
    VncKeyMappingFile1 = VC\PS2-Keyboard.dis
    VncRefreshRate1 = 500
    VncTitle1 = Debug
    ActivateSnmp = 2
    ActivateModbus = 1
    NumSlaves = -1
    NumAllBlocks = -1
    MemSizeIn = -1
    MemSizeOut = -1
  Connector IF3:
    DNAConfiguration = manual
  ConfigurationID = Static_Config1
  PermanentPvSize = 4096
  SystemTick = 5000
  IdleTaskClass = 4
  Cyclic1Duration = 5000
  Cyclic1Tolerance = 5000
  Cyclic2Duration = 10000
  Cyclic2Tolerance = 10000
  ActivateDaylightSavingTime = 1
  ActivateSntp = 1
  SntpcServAddr1 = 0.uk.pool.ntp.org
  SntpcServAddr2 = 1.uk.pool.ntp.org
  SntpcServAddr3 = 2.uk.pool.ntp.org
  SntpcServAddr4 = 3.uk.pool.ntp.org
  EthernetDefaultGateway = 172.18.219.49
  ActivateDns = 1
  DnsDefaultDomain = ukpr.local
  ActivateOpcUa = 1
  OpcUa_Security_SoftwareCertificates = 
  OpcUaInformationModels_PV_Version = 1
X20TB12a : X20TB12 v1.0.0.0
X20TB1F1 : X20TB1F v1.0.0.0
X20TB1F2 : X20TB1F v1.0.0.0
X20TB1F3 : X20TB1F v1.0.0.0
```

### IoMap.iom - X20CP1382/IoMap.iom
```iecst
VAR_CONFIG
	::operationModeWrite AT %QW."RTAC".operationModeWrite;
	::cmdOperationModeWrite AT %QX."RTAC".BlockSendOnce03;
	::OperationModeWriteACK AT %IX."RTAC".BlockSendOnceAck03;
	::RTACOperationMode AT %IW."RTAC".operationMode;
	::RTACActivePower AT %IW."RTAC".activePower;
	::RTACSoC AT %IW."RTAC".SOC;
	::DNO:DI1 AT %IX."X2a".DigitalInput01;
	::DNO:DI2 AT %IX."X2a".DigitalInput02;
	::DNO:DI3 AT %IX."X2a".DigitalInput03;
	::DNO:DO1 AT %QX."X3a".DigitalOutput01;
	::DNO:DO2 AT %QX."X3a".DigitalOutput02;
	::powerOutputDINT AT %QD."RTAC".powerWrite;
	cmdWritePowerOutput AT %QX."RTAC".BlockSendOnce01;
	WritePowerOutputACK AT %IX."RTAC".BlockSendOnceAck01;
	::Modbus:RTACModuleOK AT %IX."RTAC".ModuleOk;
	::Modbus:RTACActInternalError AT %IX."RTAC".ActInternalError;
	::Modbus:RTACActContError AT %IX."RTAC".ActConfError;
	::Modbus:RTACActOverloadError AT %IX."RTAC".ActOverloadError;
	::Modbus:RTACActModusError AT %IX."RTAC".ActModbusError;
	::Modbus:RTACActSlvConError AT %IX."RTAC".ActSlvConError;
	::Modbus:RTACActRefreshError AT %IX."RTAC".ActRefreshError;
	::Modbus:RTACModSlaveState AT %IW."RTAC".ModSlaveState;
	::Modbus:RTACModbusErrorLast AT %IW."RTAC".ModbusErrorLast;
	::Modbus:RTACLastErrBlockNr AT %IW."RTAC".LastErrBlockNr;
	::Modbus:RTACModbusErrorCnt AT %IW."RTAC".ModbusErrorCnt;
	::Modbus:RTACModbusConErrorCnt AT %IW."RTAC".ModbusConErrorCnt;
	::Modbus:RTACModbusPktRefreshTimoutCnt AT %IW."RTAC".ModbusPktRefreshTimeoutCnt;
	::Modbus:RTACPktPendPerSec AT %IW."RTAC".ModbusPktPendPerSec;
	::Modbus:RTACModbusMeanResponseTime AT %IW."RTAC".ModbusMeanResponseTime;
	::Modbus:RTACModbusSlaveDiag AT %QX."RTAC".ModbusSlaveDiag;
	::DNO_SIGNAL:Stage1_Input AT %IX."X2".DigitalInput01;
	::DNO_SIGNAL:Stage2_Input AT %IX."X2".DigitalInput02;
	::DNO_SIGNAL:G59_Input AT %IX."X2".DigitalInput03;
	::DNO_SIGNAL:Stage1_Confirmed AT %QX."X3".DigitalOutput01;
	::DNO_SIGNAL:Stage2_Confirmed AT %QX."X3".DigitalOutput02;
	::DNO_SIGNAL:TX123OPEN AT %IX."X2".DigitalInput04;
END_VAR
```

## Logical view

Binary libraries used (declarations not repeated): operator, runtime, astime, AsIecCon, standard, MTLookUp 2.00.1, sys_lib, brsystem, MTFilter 2.10.0, MTTypes 1.03.0, AsBrMath, LoopCont 3.03.2

### Global.var - Global variables
```iecst
VAR
	activePower : INT;
	cmdOperationModeWrite : BOOL;
	cmdToDynamicContainment : BOOL; (*command to turn on DC*)
	cmdToManual : BOOL; (*command to turn switch to Manual only mode*)
	cmdToStaticFFR : BOOL; (*command to turn on StaticFFR*)
	cmdTurnTestModeOff : BOOL;
	cmdTurnTestModeOn : BOOL;
	cmdWritePowerOutput : BOOL;
	durationTimer : TIME;
	DynamicContainmentEnabled : BOOL;
	expectedOutput : INT;
	frequency : UINT; (*frequency for the control*)
END_VAR
VAR CONSTANT
	GRID_FREQUENCY : REAL := 50.0;
END_VAR
VAR
	idleExpectedOutput : INT;
	injFrequency : UINT; (*injected Frequency*)
	manualFrequency : UINT; (*to inject frequency*)
	maxBatteryPower : INT;
	maxExpectedOutput : INT;
	operationModeWrite : UINT;
	OperationModeWriteACK : BOOL;
	PhaseLoss : BOOL; (*any Phase lost*)
	powerOutput : INT;
	RTACActivePower : INT;
	RTACOperationMode : UINT;
	RTACSoC : UINT;
	StaticFFREnabled : BOOL;
	staticThreshold : UINT;
	sumPhaseLoss : BOOL;
	testModeOn : BOOL; (*test mode on*)
	testModeOn1 : BOOL;
	WritePowerOutputACK : BOOL;
	DCbaselineAdjustment : INT;
	cmdToFFR : BOOL;
	diACSwitch : BOOL;
	voltPhaseA : REAL;
	voltPhaseB : REAL;
	voltPhaseC : REAL;
	curPhaseA : REAL;
	curPhaseB : REAL;
	curPhaseC : REAL;
	pf : INT;
	ManualModeEnabled : BOOL;
	powerOutputManual : INT;
	doACSwitch : BOOL;
	diPhase1LossGen : BOOL;
	aiFrequency : UINT;
	filterFreq : REAL;
	powerOutputWriteBlock : BOOL;
	controlState : UINT;
	cmdToIdle : BOOL;
	baselineAuto : BOOL;
	cmdToFluenceManual : BOOL;
	powerOutputDINT : DINT;
	baseLCCounter : LCCounter;
	DCbaselineAdjustmentManual : INT;
END_VAR
```


### Program Logical/StaticFFR (IEC)

#### Variables.var
```iecst
VAR
	timerON : BOOL;
	input : BOOL;
	output : BOOL;
	elapsedTime : TIME;
	TON_01 : TON;
	tmp : BOOL;
	prevPowerOutput : INT;
END_VAR
```

#### Cyclic.st
```iecst
PROGRAM _CYCLIC
	(* Insert code here *)
	IF StaticFFREnabled THEN
		(* call function block *)

		TON_01( IN:=timerON, PT:=durationTimer );

		IF aiFrequency <= staticThreshold AND NOT(diPhase1LossGen) AND aiFrequency > 4900 THEN
			timerON := TRUE;
		END_IF

		IF timerON AND aiFrequency > 4900 THEN
			powerOutput := maxBatteryPower;
		ELSE
			powerOutput := idleExpectedOutput;
		END_IF

		(* assign results to variables *)
		output := TON_01.Q;
		elapsedTime := TON_01.ET;

		IF timerON AND output THEN
			timerON := FALSE;
		END_IF

		doACSwitch := timerON;
		diACSwitch := timerON;
	END_IF;

END_PROGRAM
```

#### Init.st
```iecst
PROGRAM _INIT
	(* Insert code here *)
	frequency := 0;

	durationTimer := T#1800s;
	prevPowerOutput := -1;

END_PROGRAM
```

### Program Logical/DynamicContAll (IEC)

#### Cyclic.st
```iecst
PROGRAM _CYCLIC

//	IF testModeOn THEN
//
//		IF injFrequency < MIN_INJ_FREQ THEN
//			injFrequency := MIN_INJ_FREQ;
//		END_IF;
//
//		IF injFrequency > MAX_INJ_FREQ THEN
//			injFrequency := MAX_INJ_FREQ;
//		END_IF;
//
//
//		:= injFrequency;
//	ELSE
//		frequency := aiFrequency;
//	END_IF;
//
//	MovingAverage.In:= UINT_TO_REAL(frequency);
//	MovingAverage();
//
//	filterFreq := brmceil(MovingAverage.Out*10)/1000;
//	filterFreqMA := brmceil(MovingAverage.Out*10)/1000;
//
//
//	LowPassFilter.In:= UINT_TO_REAL(frequency);;
//	LowPassFilter();
//
//	filterFreqLowPass:= brmceil(LowPassFilter.Out*10)/1000;
//
//
//
//	IF DynamicContainmentEnabled THEN
//
//
//
//		IF NOT(diPhase1LossGen) THEN
//			freqDev := filterFreq - GRID_FREQUENCY;
//		ELSE
//			freqDev := 0;
//		END_IF;
//
//
//		Table.InX:= freqDev;   (* freq deviation *)
//		Table();          (* run table lookup *)
//		powerRatio:= Table.Out; (* calculated % output *)
//
//
//
//		powerOutputTmp :=  REAL_TO_INT(INT_TO_REAL(maxExpectedOutput) * powerRatio/100.00 + DCbaselineAdjustment);
//
//		diff := expected - powerOutputTmp;
//
//		error := (INT_TO_REAL(powerOutputTmp) / INT_TO_REAL(expected))*100 - 100;
//
//		powerOutputDINT := REAL_TO_DINT(INT_TO_REAL(maxExpectedOutput) * powerRatio/100.00 + DCbaselineAdjustment);
//
//		IF powerOutputDINT = 20000 THEN
//			powerOutputDINT := 20200;
//		END_IF;
//
//
//	END_IF;
//
//	IF NOT(cmdWritePowerOutput) AND NOT(WritePowerOutputACK) THEN
//
//		IF prevPowerOutput <> powerOutputDINT THEN
//			cmdWritePowerOutput := TRUE;
//		END_IF;
//		prevPowerOutput := powerOutputDINT;
//	END_IF;
//
//	IF WritePowerOutputACK THEN
//		cmdWritePowerOutput := FALSE;
//	END_IF;
//
END_PROGRAM
```

#### Init.st
```iecst
PROGRAM _INIT

    (* 1D lookup table *)
	Table.NodeVectorX[0] := -0.5;					Table.FcnValues[0] := 100;
	Table.NodeVectorX[1] := -0.2;					Table.FcnValues[1] := 5;
	Table.NodeVectorX[2] := -1*0.02;		Table.FcnValues[2] := 0.135;
	Table.NodeVectorX[3] := -1*GRID_DEADAND+0.001;	Table.FcnValues[3] := 0;
	Table.NodeVectorX[4] := GRID_DEADAND-0.001;		Table.FcnValues[4] := 0;
	//LF & HF
//	Table.NodeVectorX[5] := 0.02;			Table.FcnValues[5] := -0.135;
//	Table.NodeVectorX[6] := 0.2;					Table.FcnValues[6] := -5;
	//	Table.NodeVectorX[7] := 0.5;					Table.FcnValues[7] := -100;

	//LF Only
	Table.NodeVectorX[5] := 0.02;			Table.FcnValues[5] := 0;
	Table.NodeVectorX[6] := 0.2;					Table.FcnValues[6] := 0;
	Table.NodeVectorX[7] := 0.5;					Table.FcnValues[7] := 0;

	Table.NumberOfNodes:= 8;
	Table.Mode:= mtCONSTANT_END_VALUE;
	Table.Enable:= 1; (* enable function block *)

	MAX_INJ_FREQ := 5200;
	MIN_INJ_FREQ := 4800;

	MovingAverage.WindowLength:= 3; (* moving window length *)
	MovingAverage.Enable:= 1;

	LowPassFilter.CutOffFrequency:= 20; (* cut-off frequency [Hz] *)
	LowPassFilter.Order:= 1;             (* 3rd order low-pass filter *)
	LowPassFilter.Type:= mtBESSEL;       (* bessel filter *)
	LowPassFilter.Enable:= 1;            (* enable function block *)

	DCbaselineAdjustment := 0;

	expected := 0;

	activePower := 0;

END_PROGRAM
```

### Program Logical/DynamicContainment (IEC)

#### Variables.var
```iecst
VAR
	Table : MTLookUpTable;
	mtCONSTANT_END_VALUE : MTLookUpModeEnum;
	freqDev : REAL;
	powerOut : REAL;
	powerRatio : REAL;
END_VAR
VAR CONSTANT
	GRID_DEADAND : REAL := 0.015;
END_VAR
VAR
	freqDevUINT : UINT;
	freqDevINT : INT;
	prevPowerOutput : INT;
	MovingAverage : MTFilterMovingAverage;
	expected : INT;
	diff : INT;
	powerOutputTmp : INT;
	error : REAL;
END_VAR
```

#### Cyclic.st
```iecst
PROGRAM _CYCLIC

	IF DynamicContainmentEnabled THEN

		IF NOT(diPhase1LossGen) THEN
			freqDev := filterFreq - GRID_FREQUENCY;
		ELSE
			freqDev := 0;
		END_IF;

			Table.InX:= freqDev;   (* freq deviation *)
			Table();          (* run table lookup *)
			powerRatio:= Table.Out; (* calculated % output *)

		powerOutputTmp :=  REAL_TO_INT(INT_TO_REAL(maxExpectedOutput) * powerRatio/100.00 + DCbaselineAdjustment);

		diff := expected - powerOutputTmp;

		error := (INT_TO_REAL(powerOutputTmp) / INT_TO_REAL(expected))*100 - 100;

		powerOutputDINT := REAL_TO_DINT(INT_TO_REAL(maxExpectedOutput) * powerRatio/100.00 + DCbaselineAdjustment);

		IF powerOutputDINT = 20000 THEN
			powerOutputDINT := 20200;
		END_IF;

		IF powerOutput = 0 THEN
			powerOutput := 1;
		END_IF;

	END_IF;

END_PROGRAM
```

#### Init.st
```iecst
PROGRAM _INIT

    (* 1D lookup table *)
	Table.NodeVectorX[0] := -0.5;					Table.FcnValues[0] := 100;
	Table.NodeVectorX[1] := -0.2;					Table.FcnValues[1] := 5;
	Table.NodeVectorX[2] := -1*0.02;		Table.FcnValues[2] := 0.135;
	Table.NodeVectorX[3] := -1*GRID_DEADAND+0.001;	Table.FcnValues[3] := 0;
	Table.NodeVectorX[4] := GRID_DEADAND-0.001;		Table.FcnValues[4] := 0;
	//LF & HF
//	Table.NodeVectorX[5] := 0.02;			Table.FcnValues[5] := -0.135;
//	Table.NodeVectorX[6] := 0.2;					Table.FcnValues[6] := -5;
	//	Table.NodeVectorX[7] := 0.5;					Table.FcnValues[7] := -100;

	//LF Only
	Table.NodeVectorX[5] := 0.02;			Table.FcnValues[5] := 0;
	Table.NodeVectorX[6] := 0.2;					Table.FcnValues[6] := 0;
	Table.NodeVectorX[7] := 0.5;					Table.FcnValues[7] := 0;

	Table.NumberOfNodes:= 8;
	Table.Mode:= mtCONSTANT_END_VALUE;
	Table.Enable:= 1; (* enable function block *)

	DCbaselineAdjustment := 0;

	expected := 0;

	activePower := 0;

END_PROGRAM
```

- Visualisation Logical/Visu_Resized (not shown)

- Visualisation Logical/Visu (not shown)

### Program Logical/Main (IEC)

#### Variables.var
```iecst
VAR
	prevOperationMode : UINT;
	prevRTACOperationMode : UINT;
END_VAR
```

#### Cyclic.st
```iecst
PROGRAM _CYCLIC
	//To STATIC FFR
	IF cmdToStaticFFR THEN
		StaticFFREnabled := TRUE;
		DynamicContainmentEnabled := FALSE;
		ManualModeEnabled := FALSE;
		operationModeWrite := 2;
		controlState := 3;
		powerOutput := 0;
		cmdToStaticFFR := FALSE;
		powerOutputWriteBlock := FALSE;
	END_IF

	//To DC
	IF cmdToDynamicContainment THEN
		StaticFFREnabled := FALSE;
		DynamicContainmentEnabled := TRUE;
		ManualModeEnabled := FALSE;
		operationModeWrite := 2;
		controlState := 4;
		powerOutput := 0;
		cmdToDynamicContainment := FALSE;
		powerOutputWriteBlock := FALSE;
	END_IF

	//STATIC and DC OFF
	IF cmdToManual THEN
		StaticFFREnabled := FALSE;
		DynamicContainmentEnabled := FALSE;
		ManualModeEnabled := TRUE;
		operationModeWrite := 2;
		controlState := 2;
		powerOutputManual := 0;
		powerOutput := 0;
		cmdToManual := FALSE;
		powerOutputWriteBlock := FALSE;

	END_IF;

	//STATIC and DC OFF
	IF cmdToFluenceManual THEN
		StaticFFREnabled := FALSE;
		DynamicContainmentEnabled := FALSE;
		ManualModeEnabled := FALSE;
		operationModeWrite := 2;
		controlState := 2;
		powerOutputManual := 0;
		powerOutput := 0;
		cmdToFluenceManual := FALSE;
		powerOutputWriteBlock := TRUE;

	END_IF;

	//STATIC and DC OFF
	IF cmdToFFR THEN
		StaticFFREnabled := FALSE;
		DynamicContainmentEnabled := FALSE;
		ManualModeEnabled := FALSE;
		operationModeWrite := 28;
		controlState := 28;
		powerOutput := 0;
		cmdToFFR := FALSE;
		powerOutputWriteBlock := TRUE;

	END_IF;

	//STATIC and DC OFF
	IF cmdToIdle THEN
		StaticFFREnabled := FALSE;
		DynamicContainmentEnabled := FALSE;
		ManualModeEnabled := FALSE;
		operationModeWrite := 1;
		controlState := 1;
		powerOutput := 0;
		cmdToIdle := FALSE;
		powerOutputWriteBlock := TRUE;

	END_IF;

	IF prevRTACOperationMode <> RTACOperationMode THEN
		IF RTACOperationMode = 28 AND controlState <> 28 THEN
			cmdToFFR := TRUE;
		END_IF;

		IF RTACOperationMode = 2 AND controlState <> 4 THEN
			cmdToManual := TRUE;
		END_IF;

		IF RTACOperationMode = 1  AND controlState <> 1 THEN
			cmdToIdle := TRUE;
		END_IF;

		prevRTACOperationMode := RTACOperationMode;
	END_IF;
//
//	prevOperationMode := operationModeWrite;
//
//	IF OperationModeWriteACK THEN
//		cmdOperationModeWrite := FALSE;
//	END_IF;

	//Test Mode
	IF cmdTurnTestModeOn THEN
		testModeOn := TRUE;
		injFrequency := 5000;
		cmdTurnTestModeOn := FALSE;
	END_IF;

	IF cmdTurnTestModeOff THEN
		testModeOn := FALSE;
		cmdTurnTestModeOff := FALSE;
	END_IF;

END_PROGRAM
```

#### Init.st
```iecst
PROGRAM _INIT
	(* Insert code here *)

	RTACOperationMode := 0;
	RTACActivePower := 0;
	RTACSoC := 0;

END_PROGRAM
```

### Program Logical/IO (IEC)

#### Variables.var
```iecst
VAR
	MAX_INJ_FREQ : UINT;
	MIN_INJ_FREQ : UINT;
	avgVolt : REAL;
	avgCurrent : REAL;
	aiCurPhaseA : UINT;
	aiCurPhaseB : UINT;
	aiCurPhaseC : UINT;
	aiVoltPhaseA : UINT;
	aiVoltPhaseB : UINT;
	aiVoltPhaseC : UINT;
	curScalingFactor : REAL;
	aiPhaseCurrentGenL1 : INT;
	aiPhaseCurrentGenL2 : INT;
	aiPhaseCurrentGenL3 : INT;
	aiAverageCurrentGen : INT;
	aiLineVoltageGenL1L2 : INT;
	aiLineVoltageGenL2L3 : INT;
	aiLineVoltageGenL3L1 : INT;
	aiPhaseVoltageGenL1 : INT;
	aiPhaseVoltageGenL2 : INT;
	aiPhaseVoltageGenL3 : INT;
	aiActivePower : INT;
	aiReactivePower : INT;
	aiAparentPower : INT;
	aiAverageLineVoltage : INT;
	aiPF : INT;
	MovingAverage : MTFilterMovingAverage;
	LowPassFilter : MTFilterLowPass;
	mtBESSEL : MTFilterTypeEnum;
	filterFreqMA : REAL;
	filterFreqLowPass : REAL;
	aiLineVoltageBusL1L2 : INT;
	aiLineVoltageBusL2L3 : INT;
	aiLineVoltageBusL3L1 : INT;
	aiPhaseVoltageL1 : INT;
	aiPhaseVoltageL2 : INT;
	aiPhaseVoltageL3 : INT;
	aiLineVoltageSync1 : INT;
	aiLineVoltageSync2 : INT;
	aiFrequencySync1 : UINT;
	aiFrequencySync2 : UINT;
END_VAR
```

#### Cyclic.st
```iecst
PROGRAM _CYCLIC

	IF testModeOn THEN

		IF injFrequency < MIN_INJ_FREQ THEN
			injFrequency := MIN_INJ_FREQ;
		END_IF;

		IF injFrequency > MAX_INJ_FREQ THEN
			injFrequency := MAX_INJ_FREQ;
		END_IF;

		frequency := injFrequency;
	ELSE
		frequency := aiFrequency;
	END_IF;

	MovingAverage.In:= UINT_TO_REAL(frequency);

	MovingAverage();
	// filterFreq := MovingAverage.Out/100;
	filterFreq := brmceil(MovingAverage.Out*10)/1000;
	filterFreqMA := brmceil(MovingAverage.Out*10)/1000;

	LowPassFilter.In:= UINT_TO_REAL(frequency);;
	(* call function block *)
	LowPassFilter();
	filterFreqLowPass:= LowPassFilter.Out/100;
	LowPassFilter.Update:= 0;

	activePower := aiActivePower;

	powerOutputDINT := INT_TO_DINT(powerOutput);

END_PROGRAM
```

#### Init.st
```iecst
PROGRAM _INIT
	(* Insert code here *)
	MAX_INJ_FREQ := 5200;
	MIN_INJ_FREQ := 4800;

	MovingAverage.WindowLength:= 4; (* moving window length *)
	MovingAverage.Enable:= 1;

	LowPassFilter.CutOffFrequency:= 20; (* cut-off frequency [Hz] *)
	LowPassFilter.Order:= 3;             (* 3rd order low-pass filter *)
	LowPassFilter.Type:= mtBESSEL;       (* bessel filter *)
	LowPassFilter.Enable:= 1;            (* enable function block *)

	curScalingFactor := 1250/50;
	aiActivePower := 0;
	aiAparentPower := 0;
	aiReactivePower := 0;

	aiFrequency := 0;
	aiPF := 0;

	aiAverageLineVoltage := 0;
	aiLineVoltageGenL1L2 := 0;
	aiLineVoltageGenL2L3 := 0;
	aiLineVoltageGenL3L1 := 0;
	aiPhaseVoltageGenL1 := 0;
	aiPhaseVoltageGenL2 := 0;
	aiPhaseVoltageGenL3 := 0;

	aiAverageCurrentGen := 0;
	aiPhaseCurrentGenL1 := 0;
	aiPhaseCurrentGenL2 := 0;
	aiPhaseCurrentGenL3 := 0;

	aiLineVoltageBusL1L2 := 0;
	aiLineVoltageBusL2L3 := 0;
	aiLineVoltageBusL3L1 := 0;

	aiPhaseVoltageL1 := 0;
	aiPhaseVoltageL2 := 0;
	aiPhaseVoltageL3 := 0;

	aiLineVoltageSync1 := 0;
	aiLineVoltageSync2 := 0;

	aiFrequencySync1 := 0;
	aiFrequencySync2 := 0;

END_PROGRAM
```

### Program Logical/Settings (IEC)

#### Init.st
```iecst
PROGRAM _INIT
	maxExpectedOutput := 18000;
	idleExpectedOutput := 0;
	maxBatteryPower := 18000;
	staticThreshold := 4960;

END_PROGRAM
```

- Visualisation Logical/VisuCtrl (not shown)

### Program Logical/RTACTest (IEC)

#### Variables.var
```iecst
VAR
	prevPowerOutput : INT;
	RTACTest : BOOL;
	rampTest : BOOL;
END_VAR
```

#### Cyclic.st
```iecst
PROGRAM _CYCLIC

	IF RTACTest THEN
		IF rampTest THEN
			powerOutput := powerOutput +1;

			IF powerOutput > 1000 THEN
				powerOutput := -1000;
				END_IF;
		END_IF;
	END_IF;

END_PROGRAM
```

#### Init.st
```iecst
PROGRAM _INIT
	(* Insert code here *)
	 prevPowerOutput := -1;
END_PROGRAM
```

### Program Logical/Modbus (IEC)

#### Cyclic.st - Cyclic code
```iecst
PROGRAM _CYCLIC

	IF NOT(cmdWritePowerOutput) AND NOT(WritePowerOutputACK) THEN

		IF prevPowerOutput <> powerOutputDINT THEN
			cmdWritePowerOutput := TRUE;
		END_IF;
		prevPowerOutput := powerOutputDINT;
	END_IF;

	IF WritePowerOutputACK THEN
		cmdWritePowerOutput := FALSE;
	END_IF;

	IF NOT(cmdOperationModeWrite) AND NOT(OperationModeWriteACK) THEN
		IF prevOperationMode <> operationModeWrite THEN
			cmdOperationModeWrite := TRUE;
		END_IF;
		prevOperationMode := operationModeWrite;
	END_IF;

	IF OperationModeWriteACK THEN
		cmdOperationModeWrite := FALSE;
	END_IF;

	RTACModbusSlaveDiag := ModbusSlaveDiagOn;

END_PROGRAM
```

#### Init.st - Init code
```iecst
PROGRAM _INIT
	prevPowerOutput := -1;

	RTACModuleOK := FALSE;
	RTACActInternalError := FALSE;
	RTACActContError := FALSE;
	RTACActOverloadError := FALSE;
	RTACActModusError := FALSE;
	RTACActSlvConError := FALSE;
	RTACActRefreshError := FALSE;
	RTACModSlaveState := 0;
	RTACModbusErrorLast := 0;
	RTACLastErrBlockNr := 0;
	RTACModbusSlaveDiag := FALSE;
	RTACModbusErrorCnt := 0;
	RTACModbusConErrorCnt := 0;
	RTACModbusPktRefreshTimoutCnt := 0;
	RTACPktPendPerSec:= 0;
	RTACModbusMeanResponseTime := 0;

END_PROGRAM
```

#### Variables.var - Local variables
```iecst
VAR
	prevPowerOutput : DINT;
	prevOperationMode : UINT;
	RTACModuleOK : BOOL;
	RTACActInternalError : BOOL;
	RTACActContError : BOOL;
	RTACActOverloadError : BOOL;
	RTACActModusError : BOOL;
	RTACActSlvConError : BOOL;
	RTACActRefreshError : BOOL;
	RTACModSlaveState : UINT;
	RTACModbusErrorLast : UINT;
	RTACLastErrBlockNr : UINT;
	RTACModbusSlaveDiag : BOOL;
	RTACModbusErrorCnt : UINT;
	RTACModbusConErrorCnt : UINT;
	RTACModbusPktRefreshTimoutCnt : UINT;
	RTACPktPendPerSec : UINT;
	RTACModbusMeanResponseTime : UINT;
ModbusSlaveDiagOn : BOOL;
END_VAR
```

### Program Logical/Manual (IEC)

#### Variables.var
```iecst
VAR
	chargeToSoC : BOOL;
	chargeToSoCTarget : UINT;
	chargeToSoCPowerTarget : INT;
END_VAR
```

#### Cyclic.st
```iecst
PROGRAM _CYCLIC
	IF ManualModeEnabled THEN
		powerOutput := powerOutputManual;

		IF chargeToSoC THEN
			IF RTACSoC < chargeToSoCTarget THEN
				powerOutput := chargeToSoCPowerTarget;
			ELSE
				powerOutput := 0;
			END_IF;
		END_IF;
	END_IF;

END_PROGRAM
```

### Program Logical/DCTest (IEC)

#### Variables.var
```iecst
VAR
	sweepUp : ARRAY[0..3000] OF REAL;
	sweepDown : ARRAY[0..3000] OF REAL;
	startSweepDown : BOOL;
	out : REAL;
	ind : UINT;
	cmdStartSweepDown : BOOL;
	cmdStopSweepDown : BOOL;
	startSweepUp : BOOL;
	cmdStartSweepUp : BOOL;
	cmdStopSweepUp : BOOL;
	elapsedTime : REAL;
	stepTest : ARRAY[0..569] OF REAL;
	base1musec : UDINT;
	base100musec : UDINT;
	base1msec : UDINT;
	base100msec : UDINT;
	base1sec : UDINT;
	cmdStartStepTest : BOOL;
	startStepTest : BOOL;
	startInd : UDINT;
	prevDiff : UDINT;
	cmdStopStepTest : BOOL;
	diff : UDINT;
	sustainLF : ARRAY[0..959] OF REAL;
	startSustainLF : BOOL;
	cmdStopSustainLF : BOOL;
	cmdStartSustainLF : BOOL;
	stepTestFull : ARRAY[0..3359] OF REAL;
	sustainHF : ARRAY[0..959] OF REAL;
	cmdStartSustainHF : BOOL;
	startSustainHF : BOOL;
	cmdStopSustainHF : BOOL;
END_VAR
```

#### Cyclic.st
```iecst
PROGRAM _CYCLIC
	baseLCCounter();
	base1musec   := baseLCCounter.muscnt;
	base100musec := baseLCCounter.mus100cnt;
	base1msec    := baseLCCounter.mscnt;
	base100msec  := baseLCCounter.ms100cnt;
	base1sec     := baseLCCounter.seccnt;

	IF startSweepDown THEN
		out := sweepDown[ind];
		ind := ind + 1;
		IF ind > 3000 THEN
			cmdStopSweepDown := TRUE;
		END_IF;

	END_IF;

	IF cmdStartSweepDown THEN
		startSweepDown := TRUE;
		startSweepUp := FALSE;
		ind := 0;
		out := 50;
		cmdStartSweepDown := FALSE;
	END_IF;

	IF cmdStopSweepDown THEN
		startSweepDown := FALSE;
		ind := 0;
		out := 50;
		cmdStopSweepDown := FALSE;
	END_IF;

	IF startSweepUp THEN
		out := sweepUp[ind];
		ind := ind + 1;
		IF ind > 3000 THEN
			cmdStopSweepUp := TRUE;
		END_IF;

	END_IF;

	IF cmdStartSweepUp THEN
		startSweepDown := FALSE;
		startSweepUp := TRUE;
		ind := 0;
		out := 50;
		cmdStartSweepUp := FALSE;
	END_IF;

	IF cmdStopSweepUp THEN
		startSweepUp := FALSE;
		ind := 0;
		out := 50;
		cmdStopSweepUp := FALSE;
	END_IF;

	elapsedTime := UINT_TO_REAL(ind)/20;

	IF cmdStartStepTest THEN
		startSweepDown := FALSE;
		startSweepUp := FALSE;
		startStepTest := TRUE;
		startSustainLF := FALSE;
		startInd := base1sec;
		prevDiff := startInd;
		ind := 0;
		out := 50;
		cmdStartStepTest := FALSE;
	END_IF;

	IF cmdStopStepTest THEN
		startStepTest := FALSE;
		ind := 0;
		out := 50;
		cmdStopStepTest := FALSE;
	END_IF;

	IF startStepTest THEN

		out := stepTestFull[ind];
		diff := base1sec - startInd;

		IF prevDiff <> diff THEN
			ind := ind + 1;
			prevDiff := diff;
		END_IF;

		IF ind > 3359 THEN
//		IF ind > 60 THEN
			cmdStopStepTest := TRUE;
		END_IF;

	END_IF;

	IF cmdStartSustainLF THEN
		startSweepDown := FALSE;
		startSweepUp := FALSE;
		startStepTest := FALSE;
		startSustainLF := TRUE;
		startInd := base1sec;
		prevDiff := startInd;
		ind := 0;
		out := 50;
		cmdStartSustainLF := FALSE;
	END_IF;

	IF cmdStopSustainLF THEN
		startSustainLF := FALSE;
		ind := 0;
		out := 50;
		cmdStopSustainLF := FALSE;
	END_IF;

	IF startSustainLF THEN

		out := sustainLF[ind];
		diff := base1sec - startInd;

		IF prevDiff <> diff THEN
			ind := ind + 1;
			prevDiff := diff;
		END_IF;

		IF ind > 959 THEN
			//		IF ind > 60 THEN
			cmdStopSustainLF := TRUE;
		END_IF;

	END_IF;

	IF cmdStartSustainHF THEN
		startSweepDown := FALSE;
		startSweepUp := FALSE;
		startStepTest := FALSE;
		startSustainHF := TRUE;
		startInd := base1sec;
		prevDiff := startInd;
		ind := 0;
		out := 50;
		cmdStartSustainHF := FALSE;
	END_IF;

	IF cmdStopSustainHF THEN
		startSustainHF := FALSE;
		ind := 0;
		out := 50;
		cmdStopSustainHF := FALSE;
	END_IF;

	IF startSustainHF THEN

		out := sustainHF[ind];
		diff := base1sec - startInd;

		IF prevDiff <> diff THEN
			ind := ind + 1;
			prevDiff := diff;
		END_IF;

		IF ind > 959 THEN
			//		IF ind > 60 THEN
			cmdStopSustainHF := TRUE;
		END_IF;

	END_IF;

	IF testModeOn THEN
		injFrequency := REAL_TO_UINT(out*100);
	END_IF;

END_PROGRAM
```
